// TIA Portal project "Homework-Traffic Light" (V16)

(* hardware
DEVICE "S7-1200 station_1"  S7-1200 Station
   slot 0: "Rack_0"  S7-1200 Rack  Rack  V1.0
   slot 1: "PLC_1"  CPU 1214C DC/DC/DC  6ES7 214-1AG40-0XB0  V4.4
DEVICE "HMI_1"  KTP700 Basic PN
   slot 0: "HMI_1"  KTP700 Basic PN  6AV2 123-2GB03-0AX0  16.0.0.0
   slot 1: "HMI_RT_1"  KTP700 Basic PN  6AV2 123-2GB03-0AX0  16.0.0.0
   slot 5: "HMI_1.IE_CP_1"  PROFINET Interface  16.0.0.0
      slot 1: "PROFINET Interface_1"  PROFINET Interface
         slot 1: "Port_1"  Port
DEVICE "PC-System_1"  SIMATIC PC station
   slot 0: "SIMATIC PC station"  Rail  SIMATIC PC-Station  V1.0
      slot 125: "Stationmanager"  Station_Manager  V6.0.4
   slot 1: "HMI_RT_2"  WinCC RT Advanced  6AV2 104-0xxxx-xxxx  16.0.0.0
      slot 33792: "Computer interface"  Host interface
   slot 2: "IE general_1"  IE General  IE_CP  V8.2.0
*)

// ===== PLC "PLC_1"  CPU 1214C DC/DC/DC =====

VAR_GLOBAL   // PLC tag table "Default tag table"
   "System_Byte" AT %MB8000 : Byte;
   "FirstScan" AT %M8000.0 : Bool;
   "DiagStatusUpdate" AT %M8000.1 : Bool;
   "AlwaysTRUE" AT %M8000.2 : Bool;
   "AlwaysFALSE" AT %M8000.3 : Bool;
   "Clock_Byte" AT %MB8001 : Byte;
   "Clock_10Hz" AT %M8001.0 : Bool;
   "Clock_5Hz" AT %M8001.1 : Bool;
   "Clock_2.5Hz" AT %M8001.2 : Bool;
   "Clock_2Hz" AT %M8001.3 : Bool;
   "Clock_1.25Hz" AT %M8001.4 : Bool;
   "Clock_1Hz" AT %M8001.5 : Bool;
   "Clock_0.625Hz" AT %M8001.6 : Bool;
   "Clock_0.5Hz" AT %M8001.7 : Bool;
   "Pulse1" AT %M0.0 : Bool;
   "Pulse2" AT %M0.1 : Bool;
   "Pulse3" AT %M0.2 : Bool;
   "Pulse4" AT %M0.3 : Bool;
   "Pulse5" AT %M0.4 : Bool;
   "Pulse6" AT %M0.5 : Bool;
   "Pulse_1s" AT %M0.6 : Bool;
   "Pulse7" AT %M0.7 : Bool;
   "Remain3" AT %M1.0 : Bool;
   "Remain1" AT %M1.1 : Bool;
   "Remain2" AT %M1.2 : Bool;
   "Remain4" AT %M1.3 : Bool;
END_VAR

DATA_BLOCK "System Data"   // DB1
{ S7_Optimized_Access := 'TRUE' }
VERSION : 0.1
   VAR
      "Green A" : Bool;
      "Green B" : Bool;
      "Yellow A" : Bool;
      "Yellow B" : Bool;
      "Red A" : Bool;
      "Red B" : Bool;
      HMI_Update : Bool;
      Enable_PP1 : Bool;
      Enalbe_PP2 : Bool;
      Enalbe_PP3 : Bool;
      Start : Bool;
      Stop : Bool;
      RUN_1 : Bool;
      HMI_SET : Bool;
      "Green A _Value" : DInt;
      "Green B_Value" : DInt;
      "Yellow A_value" : DInt;
      "Yellow B_value" : DInt;
      HMI_Green_A : DInt;
      HMI_Green_B : DInt;
      HMI_Yellow_A : DInt;
      HMI_Yellow_B : DInt;
      Cancel : Bool;
      Last_signal : Bool;
      Read_Time : DTL;
      RET_Val : Word;
      Time_day : Bool;
      Time_night : Bool;
   END_VAR
BEGIN
END_DATA_BLOCK

DATA_BLOCK "7SEG_Convert1"   // DB6
{ S7_Optimized_Access := 'TRUE' }
VERSION : 0.1
// stored: InstanceOfName Convert_BCD_7SEG
"Convert_BCD_7SEG"
BEGIN
END_DATA_BLOCK

DATA_BLOCK "Data"   // DB8
{ S7_Optimized_Access := 'TRUE' }
VERSION : 0.1
   VAR
      HMI_Cancel : Bool;
      "Green A _Value" : DInt;
      "Green B_Value" : DInt;
      "1Timer_TImer" : DInt;
      "4Timer_Timer" : DInt;
      Counter_Time : DInt;
      Time_Max_Counter : DInt;
      "Yellow A_Value" : DInt;
      "Yellow B_Value" : DInt;
      "Red A_Value" : DInt;
      "Red B_Value" : DInt;
      "1Timer_Remain_LightB" : DInt;
      "1Timer_Remain_LightA" : DInt;
      TIme_LIGHT_A : DInt;
      Time_LIGHT_B : DInt;
      Timer_Light_YellowB_Remain : DInt;
      Timer_Light_YellowA_Remain : DInt;
      Counter_remain_Light_A : DInt;
      Counter_remain_Light_B : DInt;
      DEC_DIV_A : Int;
      DEC_DIV_B : Int;
      DEC_MOD_A : Int;
      DEC_MOD_B : Int;
      Remain_DEC_A : Int;
      Remain_DEC_B : Int;
      "7SEG_DIV_A" : Byte;
      "7SEG_MOD_A" : Byte;
      "7SEG_DIV_B" : Byte;
      "7SEG_MOD_B" : Byte;
   END_VAR
BEGIN
END_DATA_BLOCK

DATA_BLOCK "7SEG_Convert2"   // DB9
{ S7_Optimized_Access := 'TRUE' }
VERSION : 0.1
// stored: InstanceOfName Convert_BCD_7SEG
"Convert_BCD_7SEG"
BEGIN
END_DATA_BLOCK

DATA_BLOCK "7SEG_Convert3"   // DB10
{ S7_Optimized_Access := 'TRUE' }
VERSION : 0.1
// stored: InstanceOfName Convert_BCD_7SEG
"Convert_BCD_7SEG"
BEGIN
END_DATA_BLOCK

DATA_BLOCK "7SEG_Convert4"   // DB11
{ S7_Optimized_Access := 'TRUE' }
VERSION : 0.1
// stored: InstanceOfName Convert_BCD_7SEG
"Convert_BCD_7SEG"
BEGIN
END_DATA_BLOCK

// folder: System blocks/Program resources

DATA_BLOCK "Timer1"   // DB2
{ S7_Optimized_Access := 'TRUE' }
AUTHOR : Simatic
FAMILY : IEC
NAME : IEC_TMR
VERSION : 1.0
// stored: InstanceOfName IEC_TIMER
"IEC_TIMER"
BEGIN
END_DATA_BLOCK

DATA_BLOCK "Timer2"   // DB3
{ S7_Optimized_Access := 'TRUE' }
AUTHOR : Simatic
FAMILY : IEC
NAME : IEC_TMR
VERSION : 1.0
// stored: InstanceOfName IEC_TIMER
"IEC_TIMER"
BEGIN
END_DATA_BLOCK

DATA_BLOCK "Timer3"   // DB4
{ S7_Optimized_Access := 'TRUE' }
AUTHOR : Simatic
FAMILY : IEC
NAME : IEC_TMR
VERSION : 1.0
// stored: InstanceOfName IEC_TIMER
"IEC_TIMER"
BEGIN
END_DATA_BLOCK

DATA_BLOCK "Timer4"   // DB5
{ S7_Optimized_Access := 'TRUE' }
AUTHOR : Simatic
FAMILY : IEC
NAME : IEC_TMR
VERSION : 1.0
// stored: InstanceOfName IEC_TIMER
"IEC_TIMER"
BEGIN
END_DATA_BLOCK

DATA_BLOCK "T1"   // DB7
{ S7_Optimized_Access := 'TRUE' }
AUTHOR : Simatic
FAMILY : IEC
NAME : IEC_TMR
VERSION : 1.0
// stored: InstanceOfName IEC_TIMER
"IEC_TIMER"
BEGIN
END_DATA_BLOCK

// folder: (top level)

FUNCTION_BLOCK "Convert_BCD_7SEG"   // FB1, SCL
{ S7_Optimized_Access := 'TRUE' }
VERSION : 0.1
   VAR_INPUT
      BCD_Val : Int;
   END_VAR
   VAR_OUTPUT
      "7SEG_Val" : Byte;
   END_VAR
   VAR_TEMP
      tmp : Byte;
   END_VAR
BEGIN
   #tmp := 0;
   IF #BCD_Val =0 THEN
       #tmp := 63;
   END_IF;
   IF #BCD_Val = 1 THEN
       #tmp := 6;
   END_IF;
   IF #BCD_Val = 2 THEN
       #tmp := 91;
   END_IF;
   IF #BCD_Val = 3 THEN
       #tmp := 79;
   END_IF;
   IF #BCD_Val = 4 THEN
       #tmp := 102;
   END_IF;
   IF #BCD_Val = 5 THEN
       #tmp := 109;
   END_IF;
   IF #BCD_Val = 6 THEN
       #tmp := 125;
   END_IF;
   IF #BCD_Val = 7 THEN
       #tmp := 7;
   END_IF;
   IF #BCD_Val = 8 THEN
       #tmp := 127;
   END_IF;
   IF #BCD_Val = 9 THEN
       #tmp := 111;
   END_IF;
   #"7SEG_Val" := #tmp;
END_FUNCTION_BLOCK

FUNCTION "PP2_4Timer" : Void   // FC1, LAD
{ S7_Optimized_Access := 'TRUE' }
VERSION : 0.1
   VAR_TEMP   // added for the SCL form of the ladder/FBD networks
      _w1 : Bool;
   END_VAR
BEGIN

REGION Network 1
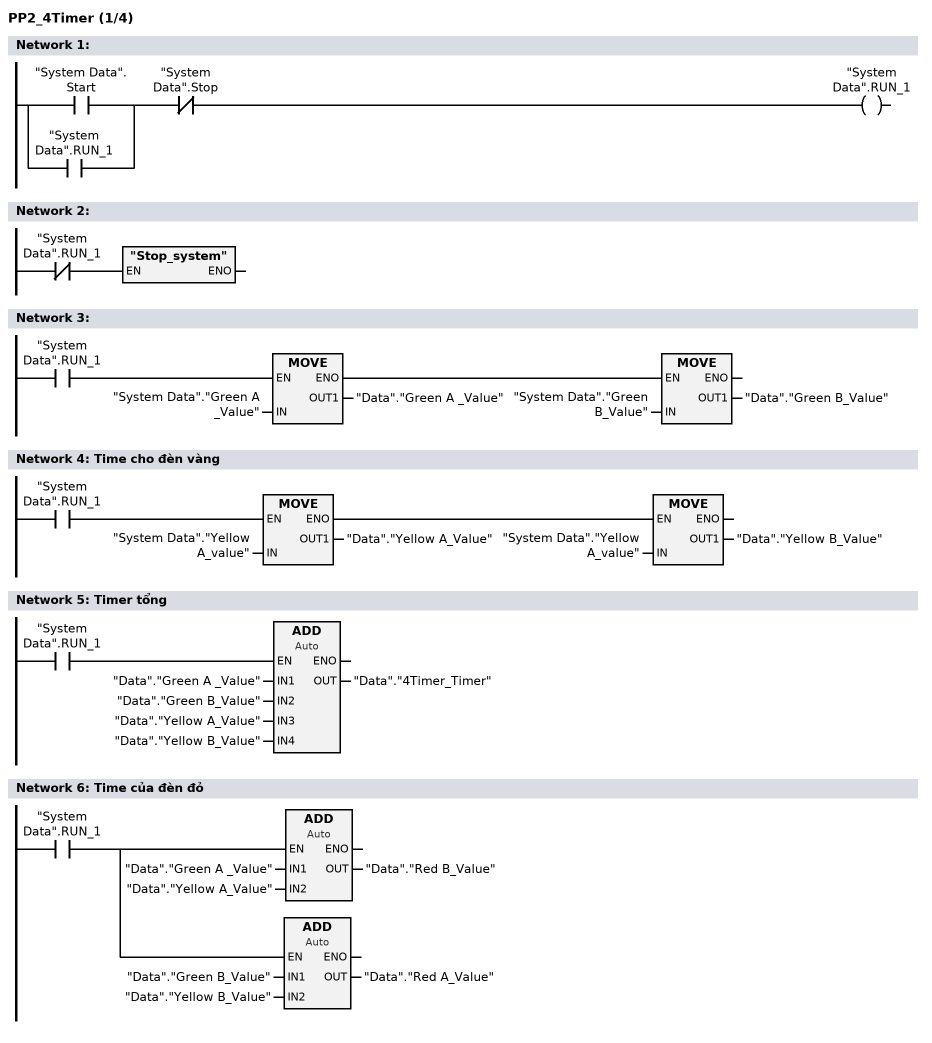
   RUNG wire#powerrail
      Contact( "System Data".Start )
      wire#w1
      I_Contact( "System Data".Stop )
      Coil( "System Data".RUN_1 )
   END_RUNG
   RUNG wire#powerrail
      Contact( "System Data".RUN_1 )
   END_RUNG wire#w1
   // the same network as SCL:
   "System Data".RUN_1 := ("System Data".Start OR "System Data".RUN_1) AND NOT "System Data".Stop;
END_REGION

REGION Network 2
   RUNG wire#powerrail
      I_Contact( "System Data".RUN_1 )
      "Stop_system"()
   END_RUNG
   // the same network as SCL:
   IF NOT "System Data".RUN_1 THEN "Stop_system"(); END_IF;
END_REGION

REGION Network 3
   RUNG wire#powerrail
      Contact( "System Data".RUN_1 )
      Move(in := "System Data"."Green A _Value", out1 => "Data"."Green A _Value")
      Move(in := "System Data"."Green B_Value", out1 => "Data"."Green B_Value")
   END_RUNG
   // the same network as SCL:
   IF "System Data".RUN_1 THEN
       "Data"."Green A _Value" := "System Data"."Green A _Value";
       "Data"."Green B_Value" := "System Data"."Green B_Value";
   END_IF;
END_REGION

REGION Network 4: Time cho đèn vàng
   RUNG wire#powerrail
      Contact( "System Data".RUN_1 )
      Move(in := "System Data"."Yellow A_value", out1 => "Data"."Yellow A_Value")
      Move(in := "System Data"."Yellow A_value", out1 => "Data"."Yellow B_Value")
   END_RUNG
   // the same network as SCL:
   IF "System Data".RUN_1 THEN
       "Data"."Yellow A_Value" := "System Data"."Yellow A_value";
       "Data"."Yellow B_Value" := "System Data"."Yellow A_value";
   END_IF;
END_REGION

REGION Network 5: Timer tổng
   RUNG wire#powerrail
      Contact( "System Data".RUN_1 )
      Add(in1 := "Data"."Green A _Value", in2 := "Data"."Green B_Value", in3 := "Data"."Yellow A_Value", in4 := "Data"."Yellow B_Value", out => "Data"."4Timer_Timer")
   END_RUNG
   // the same network as SCL:
   IF "System Data".RUN_1 THEN
       "Data"."4Timer_Timer" := "Data"."Green A _Value" + "Data"."Green B_Value" + "Data"."Yellow A_Value" + "Data"."Yellow B_Value";
   END_IF;
END_REGION

REGION Network 6: Time của đèn đỏ
   RUNG wire#powerrail
      Contact( "System Data".RUN_1 )
      wire#w1
      Add(in1 := "Data"."Green A _Value", in2 := "Data"."Yellow A_Value", out => "Data"."Red B_Value")
   END_RUNG
   RUNG wire#w1
      Add(in1 := "Data"."Green B_Value", in2 := "Data"."Yellow B_Value", out => "Data"."Red A_Value")
   END_RUNG
   // the same network as SCL:
   IF "System Data".RUN_1 THEN
       "Data"."Red B_Value" := "Data"."Green A _Value" + "Data"."Yellow A_Value";
       "Data"."Red A_Value" := "Data"."Green B_Value" + "Data"."Yellow B_Value";
   END_IF;
END_REGION

REGION Network 7
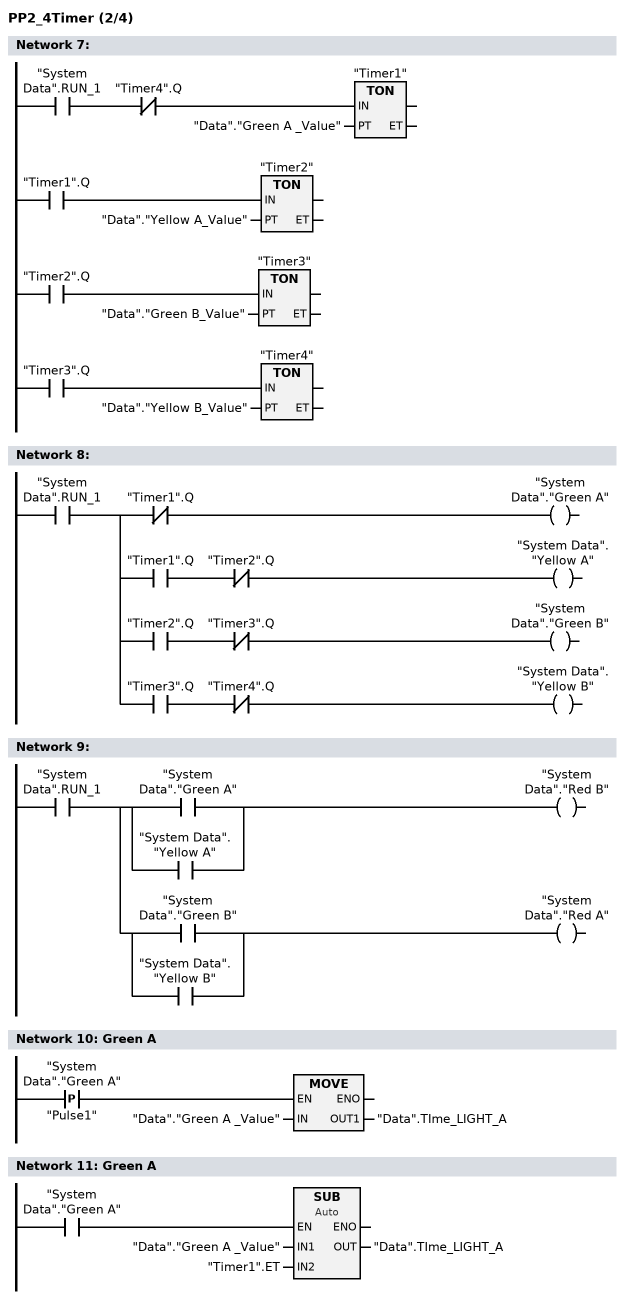
   "Timer1".TON(IN := "System Data".RUN_1 AND NOT "Timer4".Q, PT := "Data"."Green A _Value");
   "Timer2".TON(IN := "Timer1".Q, PT := "Data"."Yellow A_Value");
   "Timer3".TON(IN := "Timer2".Q, PT := "Data"."Green B_Value");
   "Timer4".TON(IN := "Timer3".Q, PT := "Data"."Yellow B_Value");
END_REGION

REGION Network 8
   RUNG wire#powerrail
      Contact( "System Data".RUN_1 )
      wire#w1
      I_Contact( "Timer1".Q )
      Coil( "System Data"."Green A" )
   END_RUNG
   RUNG wire#w1
      Contact( "Timer1".Q )
      I_Contact( "Timer2".Q )
      Coil( "System Data"."Yellow A" )
   END_RUNG
   RUNG wire#w1
      Contact( "Timer2".Q )
      I_Contact( "Timer3".Q )
      Coil( "System Data"."Green B" )
   END_RUNG
   RUNG wire#w1
      Contact( "Timer3".Q )
      I_Contact( "Timer4".Q )
      Coil( "System Data"."Yellow B" )
   END_RUNG
   // the same network as SCL:
   "System Data"."Green A" := "System Data".RUN_1 AND NOT "Timer1".Q;
   "System Data"."Yellow A" := "System Data".RUN_1 AND "Timer1".Q AND NOT "Timer2".Q;
   "System Data"."Green B" := "System Data".RUN_1 AND "Timer2".Q AND NOT "Timer3".Q;
   "System Data"."Yellow B" := "System Data".RUN_1 AND "Timer3".Q AND NOT "Timer4".Q;
END_REGION

REGION Network 9
   RUNG wire#powerrail
      Contact( "System Data".RUN_1 )
      wire#w1
      Contact( "System Data"."Green A" )
      wire#w2
      Coil( "System Data"."Red B" )
   END_RUNG
   RUNG wire#w1
      Contact( "System Data"."Yellow A" )
   END_RUNG wire#w2
   RUNG wire#w1
      Contact( "System Data"."Green B" )
      wire#w3
      Coil( "System Data"."Red A" )
   END_RUNG
   RUNG wire#w1
      Contact( "System Data"."Yellow B" )
   END_RUNG wire#w3
   // the same network as SCL:
   "System Data"."Red B" := "System Data".RUN_1 AND ("System Data"."Green A" OR "System Data"."Yellow A");
   "System Data"."Red A" := "System Data".RUN_1 AND ("System Data"."Green B" OR "System Data"."Yellow B");
END_REGION

REGION Network 10: Green A
   RUNG wire#powerrail
      P_Contact(operand := "System Data"."Green A", bit := "Pulse1")
      Move(in := "Data"."Green A _Value", out1 => "Data".TIme_LIGHT_A)
   END_RUNG
   // the same network as SCL:
   #_w1 := "System Data"."Green A" AND NOT "Pulse1";   // rising edge of "System Data"."Green A"
   "Pulse1" := "System Data"."Green A";
   IF #_w1 THEN "Data".TIme_LIGHT_A := "Data"."Green A _Value"; END_IF;
END_REGION

REGION Network 11: Green A
   RUNG wire#powerrail
      Contact( "System Data"."Green A" )
      Sub(in1 := "Data"."Green A _Value", in2 := "Timer1".ET, out => "Data".TIme_LIGHT_A)
   END_RUNG
   // the same network as SCL:
   IF "System Data"."Green A" THEN "Data".TIme_LIGHT_A := "Data"."Green A _Value" - "Timer1".ET; END_IF;
END_REGION

REGION Network 12: Yellow A
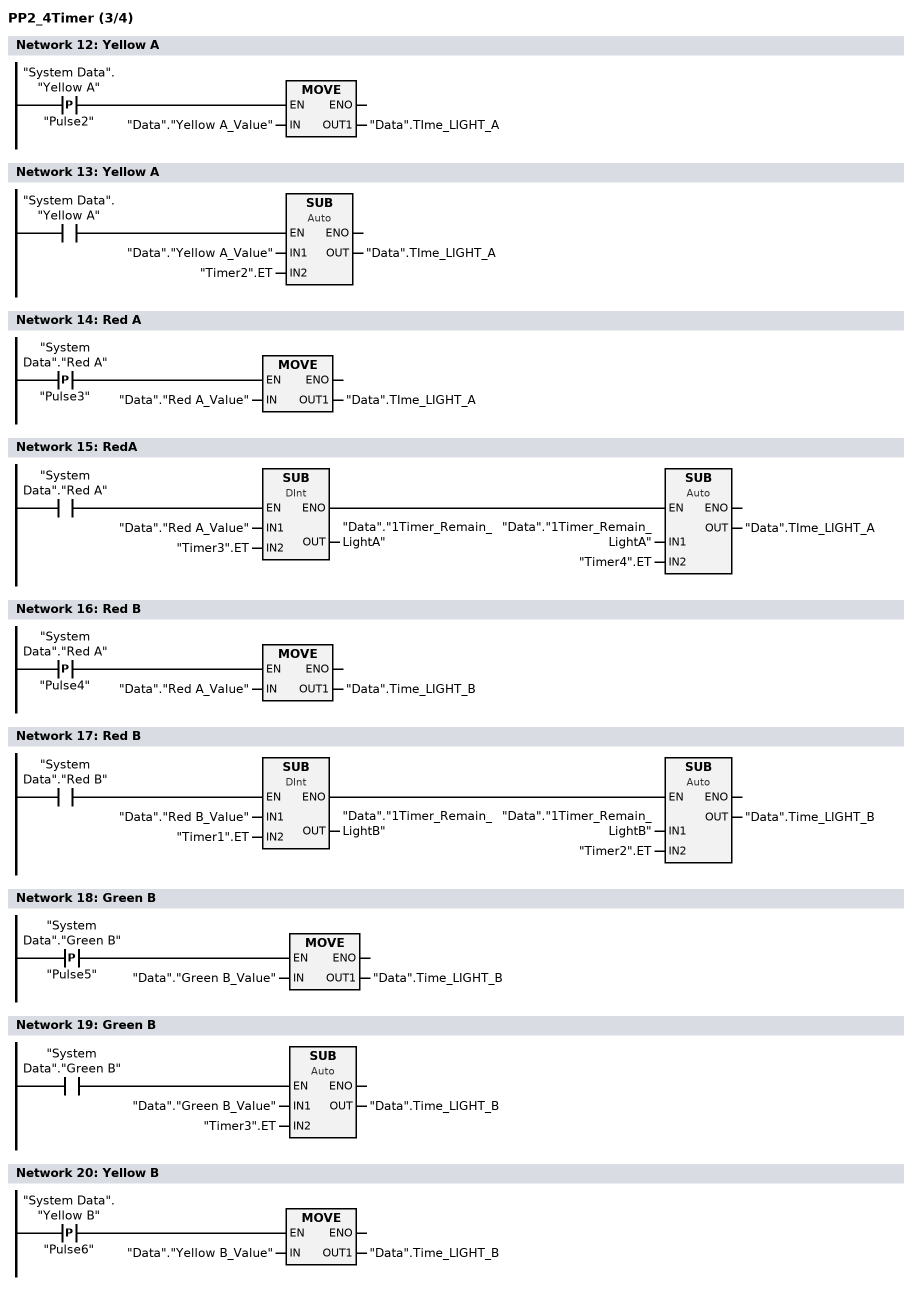
   RUNG wire#powerrail
      P_Contact(operand := "System Data"."Yellow A", bit := "Pulse2")
      Move(in := "Data"."Yellow A_Value", out1 => "Data".TIme_LIGHT_A)
   END_RUNG
   // the same network as SCL:
   #_w1 := "System Data"."Yellow A" AND NOT "Pulse2";   // rising edge of "System Data"."Yellow A"
   "Pulse2" := "System Data"."Yellow A";
   IF #_w1 THEN "Data".TIme_LIGHT_A := "Data"."Yellow A_Value"; END_IF;
END_REGION

REGION Network 13: Yellow A
   RUNG wire#powerrail
      Contact( "System Data"."Yellow A" )
      Sub(in1 := "Data"."Yellow A_Value", in2 := "Timer2".ET, out => "Data".TIme_LIGHT_A)
   END_RUNG
   // the same network as SCL:
   IF "System Data"."Yellow A" THEN "Data".TIme_LIGHT_A := "Data"."Yellow A_Value" - "Timer2".ET; END_IF;
END_REGION

REGION Network 14: Red A
   RUNG wire#powerrail
      P_Contact(operand := "System Data"."Red A", bit := "Pulse3")
      Move(in := "Data"."Red A_Value", out1 => "Data".TIme_LIGHT_A)
   END_RUNG
   // the same network as SCL:
   #_w1 := "System Data"."Red A" AND NOT "Pulse3";   // rising edge of "System Data"."Red A"
   "Pulse3" := "System Data"."Red A";
   IF #_w1 THEN "Data".TIme_LIGHT_A := "Data"."Red A_Value"; END_IF;
END_REGION

REGION Network 15: RedA
   RUNG wire#powerrail
      Contact( "System Data"."Red A" )
      { S7_Templates := "SrcType := DInt" } Sub(in1 := "Data"."Red A_Value", in2 := "Timer3".ET, out => "Data"."1Timer_Remain_LightA")
      Sub(in1 := "Data"."1Timer_Remain_LightA", in2 := "Timer4".ET, out => "Data".TIme_LIGHT_A)
   END_RUNG
   // the same network as SCL:
   IF "System Data"."Red A" THEN
       "Data"."1Timer_Remain_LightA" := "Data"."Red A_Value" - "Timer3".ET;
       "Data".TIme_LIGHT_A := "Data"."1Timer_Remain_LightA" - "Timer4".ET;
   END_IF;
END_REGION

REGION Network 16: Red B
   RUNG wire#powerrail
      P_Contact(operand := "System Data"."Red A", bit := "Pulse4")
      Move(in := "Data"."Red A_Value", out1 => "Data".Time_LIGHT_B)
   END_RUNG
   // the same network as SCL:
   #_w1 := "System Data"."Red A" AND NOT "Pulse4";   // rising edge of "System Data"."Red A"
   "Pulse4" := "System Data"."Red A";
   IF #_w1 THEN "Data".Time_LIGHT_B := "Data"."Red A_Value"; END_IF;
END_REGION

REGION Network 17: Red B
   RUNG wire#powerrail
      Contact( "System Data"."Red B" )
      { S7_Templates := "SrcType := DInt" } Sub(in1 := "Data"."Red B_Value", in2 := "Timer1".ET, out => "Data"."1Timer_Remain_LightB")
      Sub(in1 := "Data"."1Timer_Remain_LightB", in2 := "Timer2".ET, out => "Data".Time_LIGHT_B)
   END_RUNG
   // the same network as SCL:
   IF "System Data"."Red B" THEN
       "Data"."1Timer_Remain_LightB" := "Data"."Red B_Value" - "Timer1".ET;
       "Data".Time_LIGHT_B := "Data"."1Timer_Remain_LightB" - "Timer2".ET;
   END_IF;
END_REGION

REGION Network 18: Green B
   RUNG wire#powerrail
      P_Contact(operand := "System Data"."Green B", bit := "Pulse5")
      Move(in := "Data"."Green B_Value", out1 => "Data".Time_LIGHT_B)
   END_RUNG
   // the same network as SCL:
   #_w1 := "System Data"."Green B" AND NOT "Pulse5";   // rising edge of "System Data"."Green B"
   "Pulse5" := "System Data"."Green B";
   IF #_w1 THEN "Data".Time_LIGHT_B := "Data"."Green B_Value"; END_IF;
END_REGION

REGION Network 19: Green B
   RUNG wire#powerrail
      Contact( "System Data"."Green B" )
      Sub(in1 := "Data"."Green B_Value", in2 := "Timer3".ET, out => "Data".Time_LIGHT_B)
   END_RUNG
   // the same network as SCL:
   IF "System Data"."Green B" THEN "Data".Time_LIGHT_B := "Data"."Green B_Value" - "Timer3".ET; END_IF;
END_REGION

REGION Network 20: Yellow B
   RUNG wire#powerrail
      P_Contact(operand := "System Data"."Yellow B", bit := "Pulse6")
      Move(in := "Data"."Yellow B_Value", out1 => "Data".Time_LIGHT_B)
   END_RUNG
   // the same network as SCL:
   #_w1 := "System Data"."Yellow B" AND NOT "Pulse6";   // rising edge of "System Data"."Yellow B"
   "Pulse6" := "System Data"."Yellow B";
   IF #_w1 THEN "Data".Time_LIGHT_B := "Data"."Yellow B_Value"; END_IF;
END_REGION

REGION Network 21: Yellow B
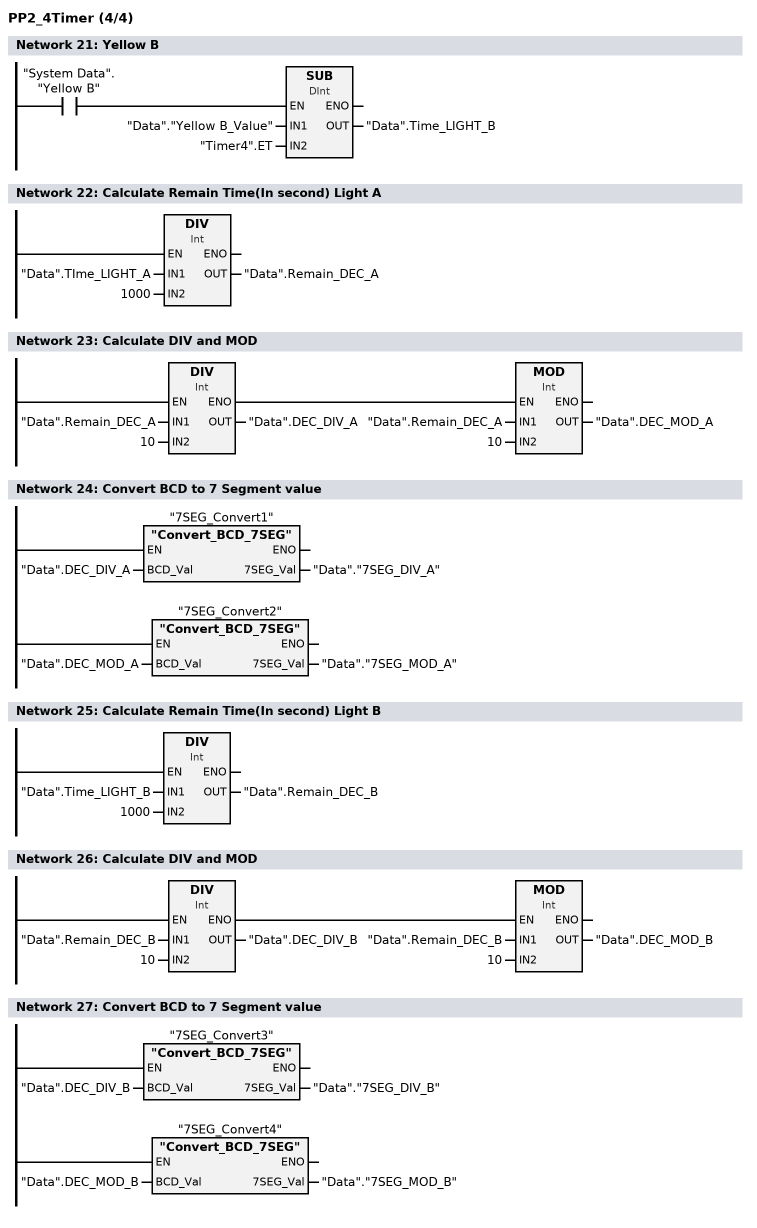
   RUNG wire#powerrail
      Contact( "System Data"."Yellow B" )
      { S7_Templates := "SrcType := DInt" } Sub(in1 := "Data"."Yellow B_Value", in2 := "Timer4".ET, out => "Data".Time_LIGHT_B)
   END_RUNG
   // the same network as SCL:
   IF "System Data"."Yellow B" THEN "Data".Time_LIGHT_B := "Data"."Yellow B_Value" - "Timer4".ET; END_IF;
END_REGION

REGION Network 22: Calculate Remain Time(In second) Light A
   RUNG wire#powerrail
      { S7_Templates := "SrcType := Int" } Div(in1 := "Data".TIme_LIGHT_A, in2 := 1000, out => "Data".Remain_DEC_A)
   END_RUNG
   // the same network as SCL:
   "Data".Remain_DEC_A := "Data".TIme_LIGHT_A / 1000;
END_REGION

REGION Network 23: Calculate DIV and MOD
   RUNG wire#powerrail
      { S7_Templates := "SrcType := Int" } Div(in1 := "Data".Remain_DEC_A, in2 := 10, out => "Data".DEC_DIV_A)
      { S7_Templates := "SrcType := Int" } Mod(in1 := "Data".Remain_DEC_A, in2 := 10, out => "Data".DEC_MOD_A)
   END_RUNG
   // the same network as SCL:
   "Data".DEC_DIV_A := "Data".Remain_DEC_A / 10;
   "Data".DEC_MOD_A := "Data".Remain_DEC_A MOD 10;
END_REGION

REGION Network 24: Convert BCD to 7 Segment value
   RUNG wire#powerrail
      "7SEG_Convert1"(BCD_Val := "Data".DEC_DIV_A, "7SEG_Val" => "Data"."7SEG_DIV_A")
   END_RUNG
   RUNG wire#powerrail
      "7SEG_Convert2"(BCD_Val := "Data".DEC_MOD_A, "7SEG_Val" => "Data"."7SEG_MOD_A")
   END_RUNG
   // the same network as SCL:
   "7SEG_Convert1"(BCD_Val := "Data".DEC_DIV_A, "7SEG_Val" => "Data"."7SEG_DIV_A");   // "Convert_BCD_7SEG"
   "7SEG_Convert2"(BCD_Val := "Data".DEC_MOD_A, "7SEG_Val" => "Data"."7SEG_MOD_A");   // "Convert_BCD_7SEG"
END_REGION

REGION Network 25: Calculate Remain Time(In second) Light B
   RUNG wire#powerrail
      { S7_Templates := "SrcType := Int" } Div(in1 := "Data".Time_LIGHT_B, in2 := 1000, out => "Data".Remain_DEC_B)
   END_RUNG
   // the same network as SCL:
   "Data".Remain_DEC_B := "Data".Time_LIGHT_B / 1000;
END_REGION

REGION Network 26: Calculate DIV and MOD
   RUNG wire#powerrail
      { S7_Templates := "SrcType := Int" } Div(in1 := "Data".Remain_DEC_B, in2 := 10, out => "Data".DEC_DIV_B)
      { S7_Templates := "SrcType := Int" } Mod(in1 := "Data".Remain_DEC_B, in2 := 10, out => "Data".DEC_MOD_B)
   END_RUNG
   // the same network as SCL:
   "Data".DEC_DIV_B := "Data".Remain_DEC_B / 10;
   "Data".DEC_MOD_B := "Data".Remain_DEC_B MOD 10;
END_REGION

REGION Network 27: Convert BCD to 7 Segment value
   RUNG wire#powerrail
      "7SEG_Convert3"(BCD_Val := "Data".DEC_DIV_B, "7SEG_Val" => "Data"."7SEG_DIV_B")
   END_RUNG
   RUNG wire#powerrail
      "7SEG_Convert4"(BCD_Val := "Data".DEC_MOD_B, "7SEG_Val" => "Data"."7SEG_MOD_B")
   END_RUNG
   // the same network as SCL:
   "7SEG_Convert3"(BCD_Val := "Data".DEC_DIV_B, "7SEG_Val" => "Data"."7SEG_DIV_B");   // "Convert_BCD_7SEG"
   "7SEG_Convert4"(BCD_Val := "Data".DEC_MOD_B, "7SEG_Val" => "Data"."7SEG_MOD_B");   // "Convert_BCD_7SEG"
END_REGION
END_FUNCTION

FUNCTION "PP1_1Timer" : Void   // FC2, LAD
{ S7_Optimized_Access := 'TRUE' }
VERSION : 0.1
   VAR_TEMP   // added for the SCL form of the ladder/FBD networks
      _w1 : Bool;
   END_VAR
BEGIN

REGION Network 1
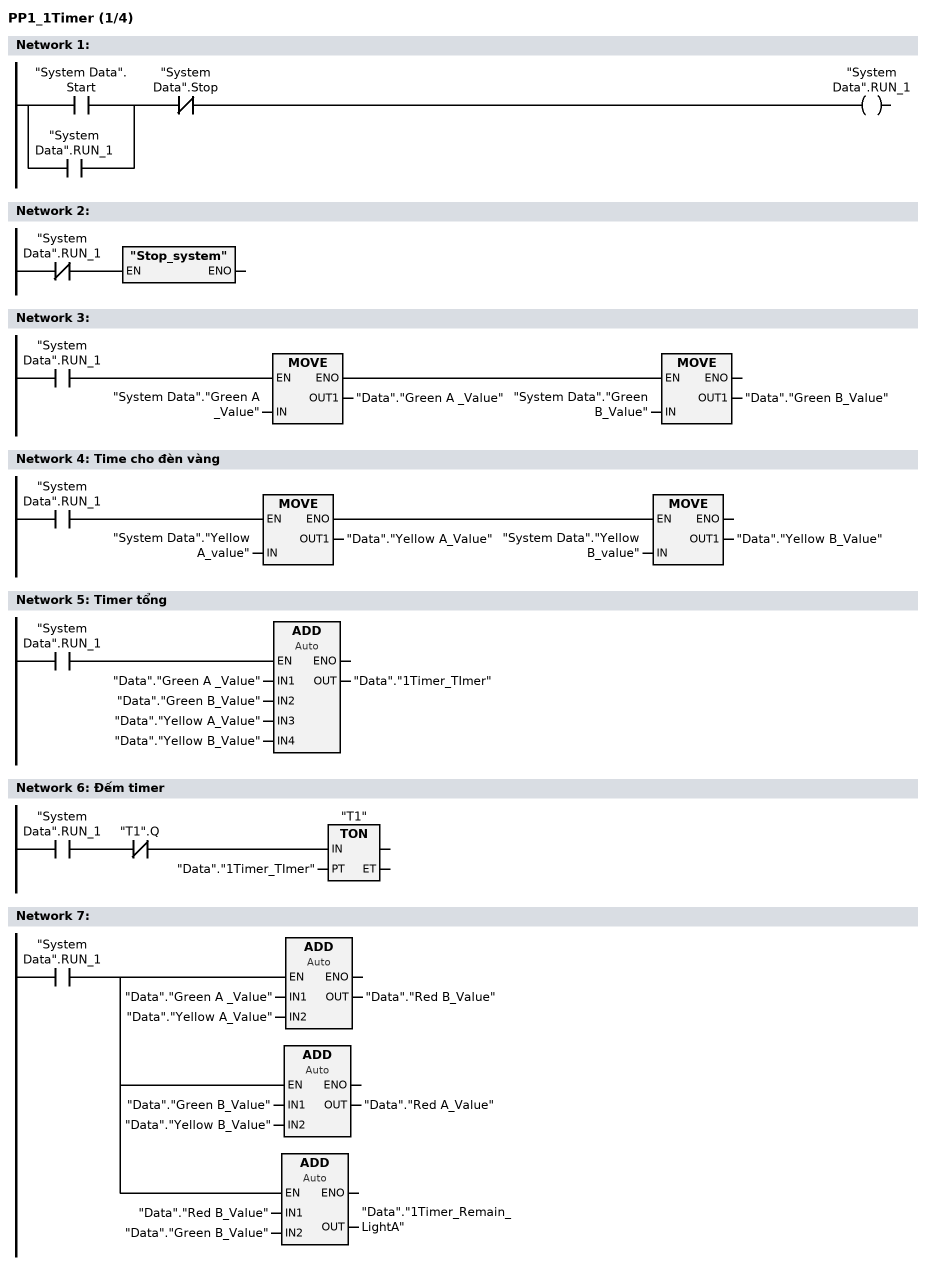
   RUNG wire#powerrail
      Contact( "System Data".Start )
      wire#w1
      I_Contact( "System Data".Stop )
      Coil( "System Data".RUN_1 )
   END_RUNG
   RUNG wire#powerrail
      Contact( "System Data".RUN_1 )
   END_RUNG wire#w1
   // the same network as SCL:
   "System Data".RUN_1 := ("System Data".Start OR "System Data".RUN_1) AND NOT "System Data".Stop;
END_REGION

REGION Network 2
   RUNG wire#powerrail
      I_Contact( "System Data".RUN_1 )
      "Stop_system"()
   END_RUNG
   // the same network as SCL:
   IF NOT "System Data".RUN_1 THEN "Stop_system"(); END_IF;
END_REGION

REGION Network 3
   RUNG wire#powerrail
      Contact( "System Data".RUN_1 )
      Move(in := "System Data"."Green A _Value", out1 => "Data"."Green A _Value")
      Move(in := "System Data"."Green B_Value", out1 => "Data"."Green B_Value")
   END_RUNG
   // the same network as SCL:
   IF "System Data".RUN_1 THEN
       "Data"."Green A _Value" := "System Data"."Green A _Value";
       "Data"."Green B_Value" := "System Data"."Green B_Value";
   END_IF;
END_REGION

REGION Network 4: Time cho đèn vàng
   RUNG wire#powerrail
      Contact( "System Data".RUN_1 )
      Move(in := "System Data"."Yellow A_value", out1 => "Data"."Yellow A_Value")
      Move(in := "System Data"."Yellow B_value", out1 => "Data"."Yellow B_Value")
   END_RUNG
   // the same network as SCL:
   IF "System Data".RUN_1 THEN
       "Data"."Yellow A_Value" := "System Data"."Yellow A_value";
       "Data"."Yellow B_Value" := "System Data"."Yellow B_value";
   END_IF;
END_REGION

REGION Network 5: Timer tổng
   RUNG wire#powerrail
      Contact( "System Data".RUN_1 )
      Add(in1 := "Data"."Green A _Value", in2 := "Data"."Green B_Value", in3 := "Data"."Yellow A_Value", in4 := "Data"."Yellow B_Value", out => "Data"."1Timer_TImer")
   END_RUNG
   // the same network as SCL:
   IF "System Data".RUN_1 THEN
       "Data"."1Timer_TImer" := "Data"."Green A _Value" + "Data"."Green B_Value" + "Data"."Yellow A_Value" + "Data"."Yellow B_Value";
   END_IF;
END_REGION

REGION Network 6: Đếm timer
   "T1".TON(IN := "System Data".RUN_1 AND NOT "T1".Q, PT := "Data"."1Timer_TImer");
END_REGION

REGION Network 7
   RUNG wire#powerrail
      Contact( "System Data".RUN_1 )
      wire#w1
      Add(in1 := "Data"."Green A _Value", in2 := "Data"."Yellow A_Value", out => "Data"."Red B_Value")
   END_RUNG
   RUNG wire#w1
      Add(in1 := "Data"."Green B_Value", in2 := "Data"."Yellow B_Value", out => "Data"."Red A_Value")
   END_RUNG
   RUNG wire#w1
      Add(in1 := "Data"."Red B_Value", in2 := "Data"."Green B_Value", out => "Data"."1Timer_Remain_LightA")
   END_RUNG
   // the same network as SCL:
   IF "System Data".RUN_1 THEN
       "Data"."Red B_Value" := "Data"."Green A _Value" + "Data"."Yellow A_Value";
       "Data"."Red A_Value" := "Data"."Green B_Value" + "Data"."Yellow B_Value";
       "Data"."1Timer_Remain_LightA" := "Data"."Red B_Value" + "Data"."Green B_Value";
   END_IF;
END_REGION

REGION Network 8
   // 5s đèn xanh
   // 5
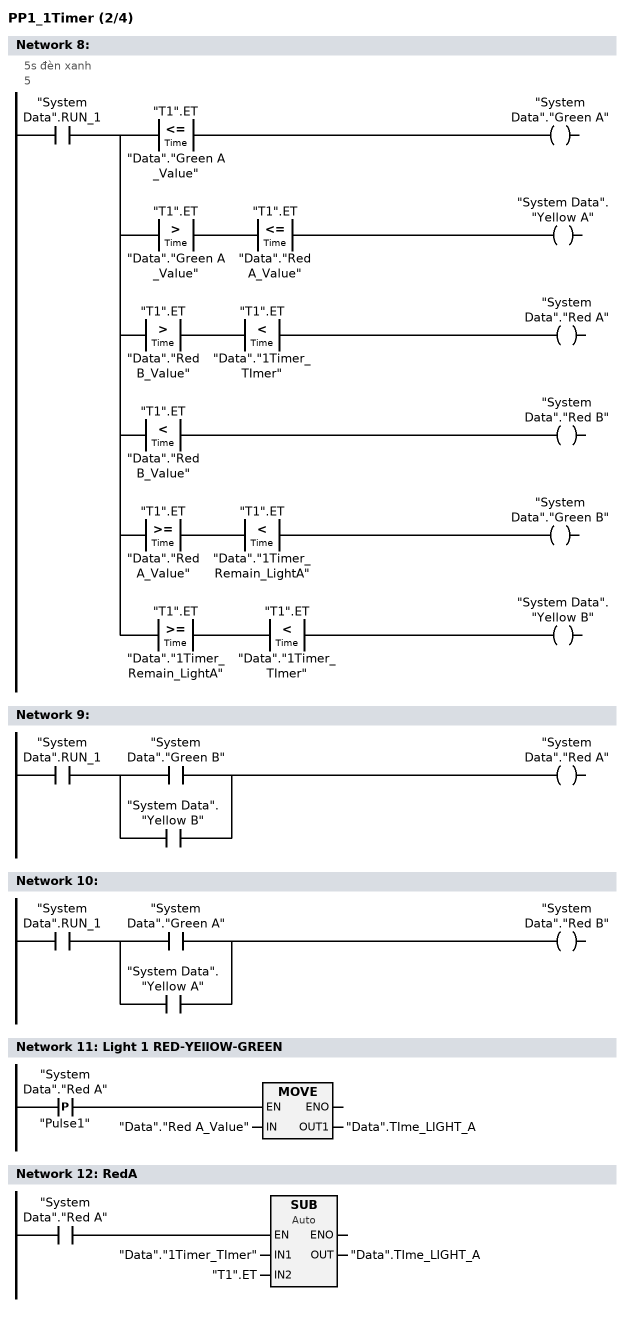
   RUNG wire#powerrail
      Contact( "System Data".RUN_1 )
      wire#w1
      { S7_Templates := "SrcType := Time" } LE_Contact(in1 := "T1".ET, in2 := "Data"."Green A _Value")
      Coil( "System Data"."Green A" )
   END_RUNG
   RUNG wire#w1
      { S7_Templates := "SrcType := Time" } GT_Contact(in1 := "T1".ET, in2 := "Data"."Green A _Value")
      { S7_Templates := "SrcType := Time" } LE_Contact(in1 := "T1".ET, in2 := "Data"."Red A_Value")
      Coil( "System Data"."Yellow A" )
   END_RUNG
   RUNG wire#w1
      { S7_Templates := "SrcType := Time" } GT_Contact(in1 := "T1".ET, in2 := "Data"."Red B_Value")
      { S7_Templates := "SrcType := Time" } LT_Contact(in1 := "T1".ET, in2 := "Data"."1Timer_TImer")
      Coil( "System Data"."Red A" )
   END_RUNG
   RUNG wire#w1
      { S7_Templates := "SrcType := Time" } LT_Contact(in1 := "T1".ET, in2 := "Data"."Red B_Value")
      Coil( "System Data"."Red B" )
   END_RUNG
   RUNG wire#w1
      { S7_Templates := "SrcType := Time" } GE_Contact(in1 := "T1".ET, in2 := "Data"."Red A_Value")
      { S7_Templates := "SrcType := Time" } LT_Contact(in1 := "T1".ET, in2 := "Data"."1Timer_Remain_LightA")
      Coil( "System Data"."Green B" )
   END_RUNG
   RUNG wire#w1
      { S7_Templates := "SrcType := Time" } GE_Contact(in1 := "T1".ET, in2 := "Data"."1Timer_Remain_LightA")
      { S7_Templates := "SrcType := Time" } LT_Contact(in1 := "T1".ET, in2 := "Data"."1Timer_TImer")
      Coil( "System Data"."Yellow B" )
   END_RUNG
   // the same network as SCL:
   "System Data"."Green A" := "System Data".RUN_1 AND ("T1".ET <= "Data"."Green A _Value");
   "System Data"."Yellow A" := "System Data".RUN_1 AND ("T1".ET > "Data"."Green A _Value") AND ("T1".ET <= "Data"."Red A_Value");
   "System Data"."Red A" := "System Data".RUN_1 AND ("T1".ET > "Data"."Red B_Value") AND ("T1".ET < "Data"."1Timer_TImer");
   "System Data"."Red B" := "System Data".RUN_1 AND ("T1".ET < "Data"."Red B_Value");
   "System Data"."Green B" := "System Data".RUN_1 AND ("T1".ET >= "Data"."Red A_Value") AND ("T1".ET < "Data"."1Timer_Remain_LightA");
   "System Data"."Yellow B" := "System Data".RUN_1 AND ("T1".ET >= "Data"."1Timer_Remain_LightA") AND ("T1".ET < "Data"."1Timer_TImer");
END_REGION

REGION Network 9
   RUNG wire#powerrail
      Contact( "System Data".RUN_1 )
      wire#w1
      Contact( "System Data"."Green B" )
      wire#w2
      Coil( "System Data"."Red A" )
   END_RUNG
   RUNG wire#w1
      Contact( "System Data"."Yellow B" )
   END_RUNG wire#w2
   // the same network as SCL:
   "System Data"."Red A" := "System Data".RUN_1 AND ("System Data"."Green B" OR "System Data"."Yellow B");
END_REGION

REGION Network 10
   RUNG wire#powerrail
      Contact( "System Data".RUN_1 )
      wire#w1
      Contact( "System Data"."Green A" )
      wire#w2
      Coil( "System Data"."Red B" )
   END_RUNG
   RUNG wire#w1
      Contact( "System Data"."Yellow A" )
   END_RUNG wire#w2
   // the same network as SCL:
   "System Data"."Red B" := "System Data".RUN_1 AND ("System Data"."Green A" OR "System Data"."Yellow A");
END_REGION

REGION Network 11: Light 1 RED-YEllOW-GREEN
   RUNG wire#powerrail
      P_Contact(operand := "System Data"."Red A", bit := "Pulse1")
      Move(in := "Data"."Red A_Value", out1 => "Data".TIme_LIGHT_A)
   END_RUNG
   // the same network as SCL:
   #_w1 := "System Data"."Red A" AND NOT "Pulse1";   // rising edge of "System Data"."Red A"
   "Pulse1" := "System Data"."Red A";
   IF #_w1 THEN "Data".TIme_LIGHT_A := "Data"."Red A_Value"; END_IF;
END_REGION

REGION Network 12: RedA
   RUNG wire#powerrail
      Contact( "System Data"."Red A" )
      Sub(in1 := "Data"."1Timer_TImer", in2 := "T1".ET, out => "Data".TIme_LIGHT_A)
   END_RUNG
   // the same network as SCL:
   IF "System Data"."Red A" THEN "Data".TIme_LIGHT_A := "Data"."1Timer_TImer" - "T1".ET; END_IF;
END_REGION

REGION Network 13
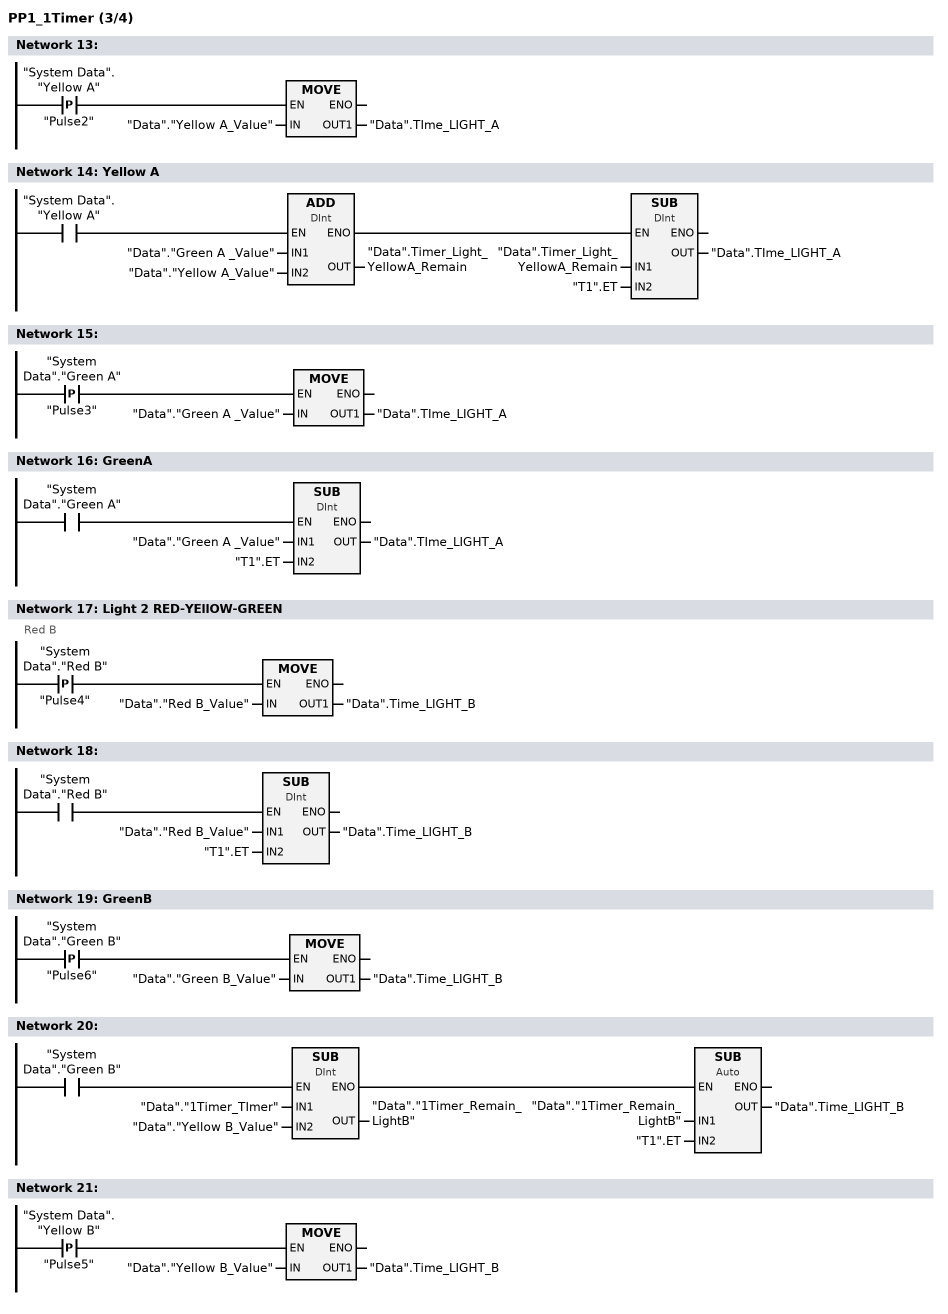
   RUNG wire#powerrail
      P_Contact(operand := "System Data"."Yellow A", bit := "Pulse2")
      Move(in := "Data"."Yellow A_Value", out1 => "Data".TIme_LIGHT_A)
   END_RUNG
   // the same network as SCL:
   #_w1 := "System Data"."Yellow A" AND NOT "Pulse2";   // rising edge of "System Data"."Yellow A"
   "Pulse2" := "System Data"."Yellow A";
   IF #_w1 THEN "Data".TIme_LIGHT_A := "Data"."Yellow A_Value"; END_IF;
END_REGION

REGION Network 14: Yellow A
   RUNG wire#powerrail
      Contact( "System Data"."Yellow A" )
      { S7_Templates := "SrcType := DInt" } Add(in1 := "Data"."Green A _Value", in2 := "Data"."Yellow A_Value", out => "Data".Timer_Light_YellowA_Remain)
      { S7_Templates := "SrcType := DInt" } Sub(in1 := "Data".Timer_Light_YellowA_Remain, in2 := "T1".ET, out => "Data".TIme_LIGHT_A)
   END_RUNG
   // the same network as SCL:
   IF "System Data"."Yellow A" THEN
       "Data".Timer_Light_YellowA_Remain := "Data"."Green A _Value" + "Data"."Yellow A_Value";
       "Data".TIme_LIGHT_A := "Data".Timer_Light_YellowA_Remain - "T1".ET;
   END_IF;
END_REGION

REGION Network 15
   RUNG wire#powerrail
      P_Contact(operand := "System Data"."Green A", bit := "Pulse3")
      Move(in := "Data"."Green A _Value", out1 => "Data".TIme_LIGHT_A)
   END_RUNG
   // the same network as SCL:
   #_w1 := "System Data"."Green A" AND NOT "Pulse3";   // rising edge of "System Data"."Green A"
   "Pulse3" := "System Data"."Green A";
   IF #_w1 THEN "Data".TIme_LIGHT_A := "Data"."Green A _Value"; END_IF;
END_REGION

REGION Network 16: GreenA
   RUNG wire#powerrail
      Contact( "System Data"."Green A" )
      { S7_Templates := "SrcType := DInt" } Sub(in1 := "Data"."Green A _Value", in2 := "T1".ET, out => "Data".TIme_LIGHT_A)
   END_RUNG
   // the same network as SCL:
   IF "System Data"."Green A" THEN "Data".TIme_LIGHT_A := "Data"."Green A _Value" - "T1".ET; END_IF;
END_REGION

REGION Network 17: Light 2 RED-YEllOW-GREEN
   // Red B
   RUNG wire#powerrail
      P_Contact(operand := "System Data"."Red B", bit := "Pulse4")
      Move(in := "Data"."Red B_Value", out1 => "Data".Time_LIGHT_B)
   END_RUNG
   // the same network as SCL:
   #_w1 := "System Data"."Red B" AND NOT "Pulse4";   // rising edge of "System Data"."Red B"
   "Pulse4" := "System Data"."Red B";
   IF #_w1 THEN "Data".Time_LIGHT_B := "Data"."Red B_Value"; END_IF;
END_REGION

REGION Network 18
   RUNG wire#powerrail
      Contact( "System Data"."Red B" )
      { S7_Templates := "SrcType := DInt" } Sub(in1 := "Data"."Red B_Value", in2 := "T1".ET, out => "Data".Time_LIGHT_B)
   END_RUNG
   // the same network as SCL:
   IF "System Data"."Red B" THEN "Data".Time_LIGHT_B := "Data"."Red B_Value" - "T1".ET; END_IF;
END_REGION

REGION Network 19: GreenB
   RUNG wire#powerrail
      P_Contact(operand := "System Data"."Green B", bit := "Pulse6")
      Move(in := "Data"."Green B_Value", out1 => "Data".Time_LIGHT_B)
   END_RUNG
   // the same network as SCL:
   #_w1 := "System Data"."Green B" AND NOT "Pulse6";   // rising edge of "System Data"."Green B"
   "Pulse6" := "System Data"."Green B";
   IF #_w1 THEN "Data".Time_LIGHT_B := "Data"."Green B_Value"; END_IF;
END_REGION

REGION Network 20
   RUNG wire#powerrail
      Contact( "System Data"."Green B" )
      { S7_Templates := "SrcType := DInt" } Sub(in1 := "Data"."1Timer_TImer", in2 := "Data"."Yellow B_Value", out => "Data"."1Timer_Remain_LightB")
      Sub(in1 := "Data"."1Timer_Remain_LightB", in2 := "T1".ET, out => "Data".Time_LIGHT_B)
   END_RUNG
   // the same network as SCL:
   IF "System Data"."Green B" THEN
       "Data"."1Timer_Remain_LightB" := "Data"."1Timer_TImer" - "Data"."Yellow B_Value";
       "Data".Time_LIGHT_B := "Data"."1Timer_Remain_LightB" - "T1".ET;
   END_IF;
END_REGION

REGION Network 21
   RUNG wire#powerrail
      P_Contact(operand := "System Data"."Yellow B", bit := "Pulse5")
      Move(in := "Data"."Yellow B_Value", out1 => "Data".Time_LIGHT_B)
   END_RUNG
   // the same network as SCL:
   #_w1 := "System Data"."Yellow B" AND NOT "Pulse5";   // rising edge of "System Data"."Yellow B"
   "Pulse5" := "System Data"."Yellow B";
   IF #_w1 THEN "Data".Time_LIGHT_B := "Data"."Yellow B_Value"; END_IF;
END_REGION

REGION Network 22: Yellow B
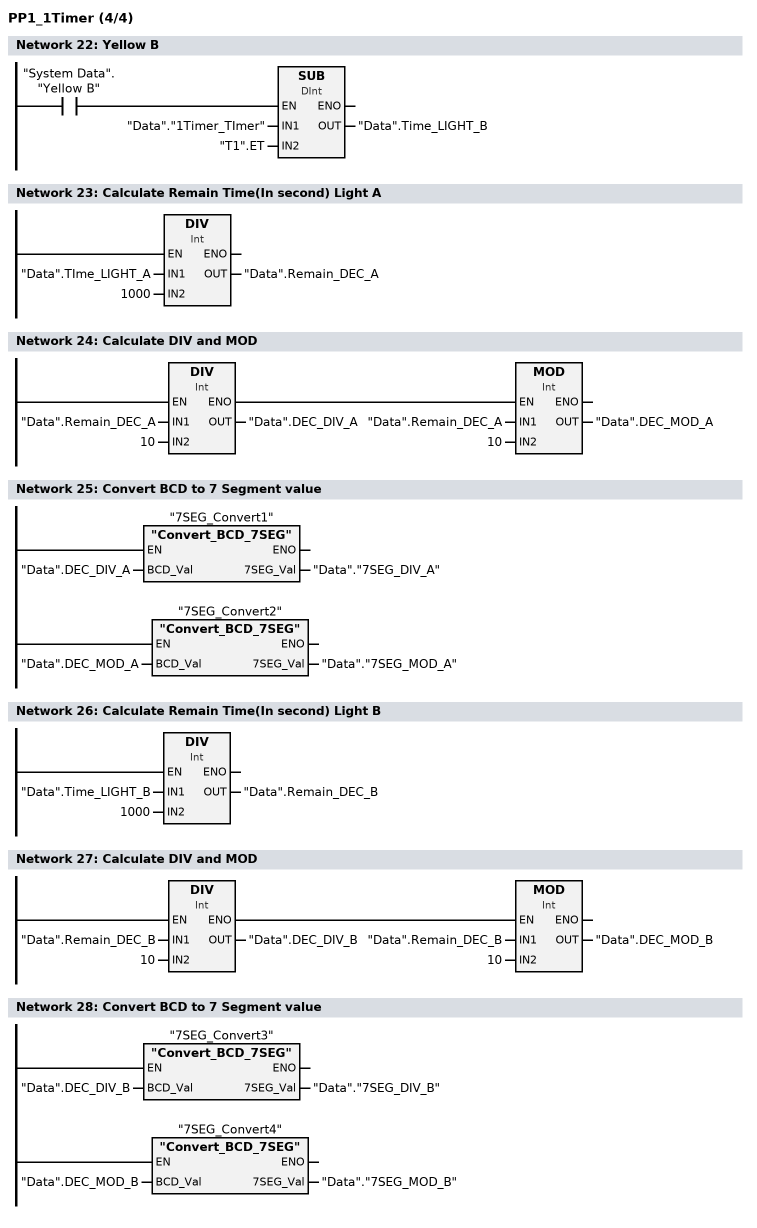
   RUNG wire#powerrail
      Contact( "System Data"."Yellow B" )
      { S7_Templates := "SrcType := DInt" } Sub(in1 := "Data"."1Timer_TImer", in2 := "T1".ET, out => "Data".Time_LIGHT_B)
   END_RUNG
   // the same network as SCL:
   IF "System Data"."Yellow B" THEN "Data".Time_LIGHT_B := "Data"."1Timer_TImer" - "T1".ET; END_IF;
END_REGION

REGION Network 23: Calculate Remain Time(In second) Light A
   RUNG wire#powerrail
      { S7_Templates := "SrcType := Int" } Div(in1 := "Data".TIme_LIGHT_A, in2 := 1000, out => "Data".Remain_DEC_A)
   END_RUNG
   // the same network as SCL:
   "Data".Remain_DEC_A := "Data".TIme_LIGHT_A / 1000;
END_REGION

REGION Network 24: Calculate DIV and MOD
   RUNG wire#powerrail
      { S7_Templates := "SrcType := Int" } Div(in1 := "Data".Remain_DEC_A, in2 := 10, out => "Data".DEC_DIV_A)
      { S7_Templates := "SrcType := Int" } Mod(in1 := "Data".Remain_DEC_A, in2 := 10, out => "Data".DEC_MOD_A)
   END_RUNG
   // the same network as SCL:
   "Data".DEC_DIV_A := "Data".Remain_DEC_A / 10;
   "Data".DEC_MOD_A := "Data".Remain_DEC_A MOD 10;
END_REGION

REGION Network 25: Convert BCD to 7 Segment value
   RUNG wire#powerrail
      "7SEG_Convert1"(BCD_Val := "Data".DEC_DIV_A, "7SEG_Val" => "Data"."7SEG_DIV_A")
   END_RUNG
   RUNG wire#powerrail
      "7SEG_Convert2"(BCD_Val := "Data".DEC_MOD_A, "7SEG_Val" => "Data"."7SEG_MOD_A")
   END_RUNG
   // the same network as SCL:
   "7SEG_Convert1"(BCD_Val := "Data".DEC_DIV_A, "7SEG_Val" => "Data"."7SEG_DIV_A");   // "Convert_BCD_7SEG"
   "7SEG_Convert2"(BCD_Val := "Data".DEC_MOD_A, "7SEG_Val" => "Data"."7SEG_MOD_A");   // "Convert_BCD_7SEG"
END_REGION

REGION Network 26: Calculate Remain Time(In second) Light B
   RUNG wire#powerrail
      { S7_Templates := "SrcType := Int" } Div(in1 := "Data".Time_LIGHT_B, in2 := 1000, out => "Data".Remain_DEC_B)
   END_RUNG
   // the same network as SCL:
   "Data".Remain_DEC_B := "Data".Time_LIGHT_B / 1000;
END_REGION

REGION Network 27: Calculate DIV and MOD
   RUNG wire#powerrail
      { S7_Templates := "SrcType := Int" } Div(in1 := "Data".Remain_DEC_B, in2 := 10, out => "Data".DEC_DIV_B)
      { S7_Templates := "SrcType := Int" } Mod(in1 := "Data".Remain_DEC_B, in2 := 10, out => "Data".DEC_MOD_B)
   END_RUNG
   // the same network as SCL:
   "Data".DEC_DIV_B := "Data".Remain_DEC_B / 10;
   "Data".DEC_MOD_B := "Data".Remain_DEC_B MOD 10;
END_REGION

REGION Network 28: Convert BCD to 7 Segment value
   RUNG wire#powerrail
      "7SEG_Convert3"(BCD_Val := "Data".DEC_DIV_B, "7SEG_Val" => "Data"."7SEG_DIV_B")
   END_RUNG
   RUNG wire#powerrail
      "7SEG_Convert4"(BCD_Val := "Data".DEC_MOD_B, "7SEG_Val" => "Data"."7SEG_MOD_B")
   END_RUNG
   // the same network as SCL:
   "7SEG_Convert3"(BCD_Val := "Data".DEC_DIV_B, "7SEG_Val" => "Data"."7SEG_DIV_B");   // "Convert_BCD_7SEG"
   "7SEG_Convert4"(BCD_Val := "Data".DEC_MOD_B, "7SEG_Val" => "Data"."7SEG_MOD_B");   // "Convert_BCD_7SEG"
END_REGION
END_FUNCTION

FUNCTION "PP3_Counter" : Void   // FC3, LAD
{ S7_Optimized_Access := 'TRUE' }
VERSION : 0.1
   VAR_TEMP   // added for the SCL form of the ladder/FBD networks
      _w1 : Bool;
   END_VAR
BEGIN

REGION Network 1: System
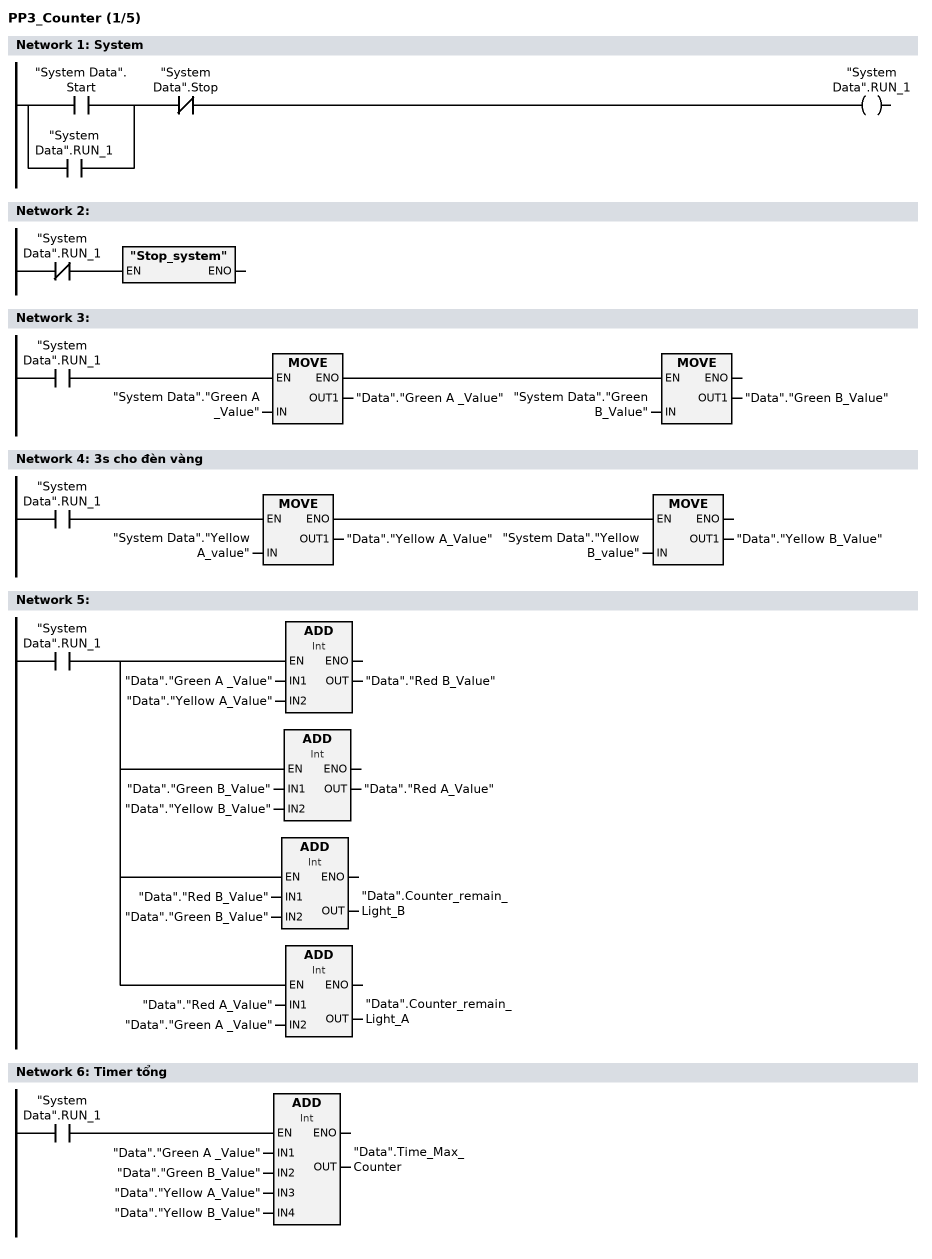
   RUNG wire#powerrail
      Contact( "System Data".Start )
      wire#w1
      I_Contact( "System Data".Stop )
      Coil( "System Data".RUN_1 )
   END_RUNG
   RUNG wire#powerrail
      Contact( "System Data".RUN_1 )
   END_RUNG wire#w1
   // the same network as SCL:
   "System Data".RUN_1 := ("System Data".Start OR "System Data".RUN_1) AND NOT "System Data".Stop;
END_REGION

REGION Network 2
   RUNG wire#powerrail
      I_Contact( "System Data".RUN_1 )
      "Stop_system"()
   END_RUNG
   // the same network as SCL:
   IF NOT "System Data".RUN_1 THEN "Stop_system"(); END_IF;
END_REGION

REGION Network 3
   RUNG wire#powerrail
      Contact( "System Data".RUN_1 )
      Move(in := "System Data"."Green A _Value", out1 => "Data"."Green A _Value")
      Move(in := "System Data"."Green B_Value", out1 => "Data"."Green B_Value")
   END_RUNG
   // the same network as SCL:
   IF "System Data".RUN_1 THEN
       "Data"."Green A _Value" := "System Data"."Green A _Value";
       "Data"."Green B_Value" := "System Data"."Green B_Value";
   END_IF;
END_REGION

REGION Network 4: 3s cho đèn vàng
   RUNG wire#powerrail
      Contact( "System Data".RUN_1 )
      Move(in := "System Data"."Yellow A_value", out1 => "Data"."Yellow A_Value")
      Move(in := "System Data"."Yellow B_value", out1 => "Data"."Yellow B_Value")
   END_RUNG
   // the same network as SCL:
   IF "System Data".RUN_1 THEN
       "Data"."Yellow A_Value" := "System Data"."Yellow A_value";
       "Data"."Yellow B_Value" := "System Data"."Yellow B_value";
   END_IF;
END_REGION

REGION Network 5
   RUNG wire#powerrail
      Contact( "System Data".RUN_1 )
      wire#w1
      { S7_Templates := "SrcType := Int" } Add(in1 := "Data"."Green A _Value", in2 := "Data"."Yellow A_Value", out => "Data"."Red B_Value")
   END_RUNG
   RUNG wire#w1
      { S7_Templates := "SrcType := Int" } Add(in1 := "Data"."Green B_Value", in2 := "Data"."Yellow B_Value", out => "Data"."Red A_Value")
   END_RUNG
   RUNG wire#w1
      { S7_Templates := "SrcType := Int" } Add(in1 := "Data"."Red B_Value", in2 := "Data"."Green B_Value", out => "Data".Counter_remain_Light_B)
   END_RUNG
   RUNG wire#w1
      { S7_Templates := "SrcType := Int" } Add(in1 := "Data"."Red A_Value", in2 := "Data"."Green A _Value", out => "Data".Counter_remain_Light_A)
   END_RUNG
   // the same network as SCL:
   IF "System Data".RUN_1 THEN
       "Data"."Red B_Value" := "Data"."Green A _Value" + "Data"."Yellow A_Value";
       "Data"."Red A_Value" := "Data"."Green B_Value" + "Data"."Yellow B_Value";
       "Data".Counter_remain_Light_B := "Data"."Red B_Value" + "Data"."Green B_Value";
       "Data".Counter_remain_Light_A := "Data"."Red A_Value" + "Data"."Green A _Value";
   END_IF;
END_REGION

REGION Network 6: Timer tổng
   RUNG wire#powerrail
      Contact( "System Data".RUN_1 )
      { S7_Templates := "SrcType := Int" } Add(in1 := "Data"."Green A _Value", in2 := "Data"."Green B_Value", in3 := "Data"."Yellow A_Value", in4 := "Data"."Yellow B_Value", out => "Data".Time_Max_Counter)
   END_RUNG
   // the same network as SCL:
   IF "System Data".RUN_1 THEN
       "Data".Time_Max_Counter := "Data"."Green A _Value" + "Data"."Green B_Value" + "Data"."Yellow A_Value" + "Data"."Yellow B_Value";
   END_IF;
END_REGION

REGION Network 7: Tạo xung 1s
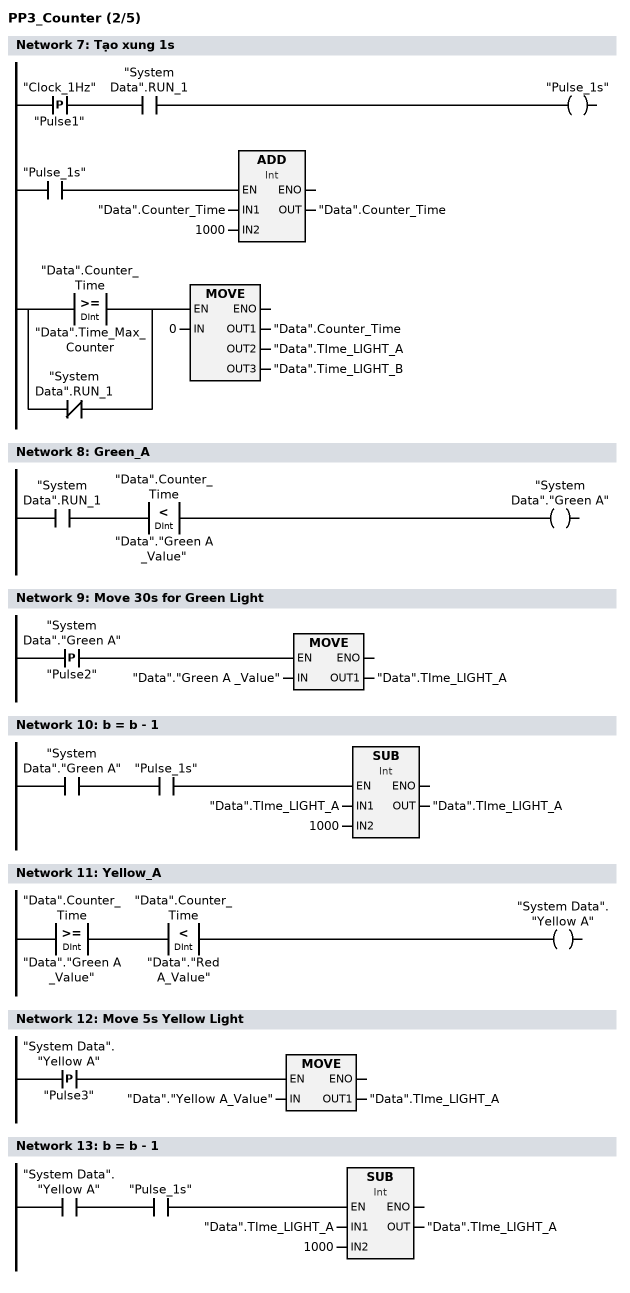
   RUNG wire#powerrail
      P_Contact(operand := "Clock_1Hz", bit := "Pulse1")
      Contact( "System Data".RUN_1 )
      Coil( "Pulse_1s" )
   END_RUNG
   RUNG wire#powerrail
      Contact( "Pulse_1s" )
      { S7_Templates := "SrcType := Int" } Add(in1 := "Data".Counter_Time, in2 := 1000, out => "Data".Counter_Time)
   END_RUNG
   RUNG wire#powerrail
      { S7_Templates := "SrcType := DInt" } GE_Contact(in1 := "Data".Counter_Time, in2 := "Data".Time_Max_Counter)
      wire#w1
      Move(in := 0, out1 => "Data".Counter_Time, out2 => "Data".TIme_LIGHT_A, out3 => "Data".Time_LIGHT_B)
   END_RUNG
   RUNG wire#powerrail
      I_Contact( "System Data".RUN_1 )
   END_RUNG wire#w1
   // the same network as SCL:
   #_w1 := "Clock_1Hz" AND NOT "Pulse1";   // rising edge of "Clock_1Hz"
   "Pulse1" := "Clock_1Hz";
   "Pulse_1s" := #_w1 AND "System Data".RUN_1;
   IF "Pulse_1s" THEN "Data".Counter_Time := "Data".Counter_Time + 1000; END_IF;
   IF ("Data".Counter_Time >= "Data".Time_Max_Counter) OR NOT "System Data".RUN_1 THEN
       "Data".Counter_Time := 0;
       "Data".TIme_LIGHT_A := 0;
       "Data".Time_LIGHT_B := 0;
   END_IF;
END_REGION

REGION Network 8: Green_A
   RUNG wire#powerrail
      Contact( "System Data".RUN_1 )
      { S7_Templates := "SrcType := DInt" } LT_Contact(in1 := "Data".Counter_Time, in2 := "Data"."Green A _Value")
      Coil( "System Data"."Green A" )
   END_RUNG
   // the same network as SCL:
   "System Data"."Green A" := "System Data".RUN_1 AND ("Data".Counter_Time < "Data"."Green A _Value");
END_REGION

REGION Network 9: Move 30s for Green Light
   RUNG wire#powerrail
      P_Contact(operand := "System Data"."Green A", bit := "Pulse2")
      Move(in := "Data"."Green A _Value", out1 => "Data".TIme_LIGHT_A)
   END_RUNG
   // the same network as SCL:
   #_w1 := "System Data"."Green A" AND NOT "Pulse2";   // rising edge of "System Data"."Green A"
   "Pulse2" := "System Data"."Green A";
   IF #_w1 THEN "Data".TIme_LIGHT_A := "Data"."Green A _Value"; END_IF;
END_REGION

REGION Network 10: b = b - 1
   RUNG wire#powerrail
      Contact( "System Data"."Green A" )
      Contact( "Pulse_1s" )
      { S7_Templates := "SrcType := Int" } Sub(in1 := "Data".TIme_LIGHT_A, in2 := 1000, out => "Data".TIme_LIGHT_A)
   END_RUNG
   // the same network as SCL:
   IF "System Data"."Green A" AND "Pulse_1s" THEN "Data".TIme_LIGHT_A := "Data".TIme_LIGHT_A - 1000; END_IF;
END_REGION

REGION Network 11: Yellow_A
   RUNG wire#powerrail
      { S7_Templates := "SrcType := DInt" } GE_Contact(in1 := "Data".Counter_Time, in2 := "Data"."Green A _Value")
      { S7_Templates := "SrcType := DInt" } LT_Contact(in1 := "Data".Counter_Time, in2 := "Data"."Red A_Value")
      Coil( "System Data"."Yellow A" )
   END_RUNG
   // the same network as SCL:
   "System Data"."Yellow A" := ("Data".Counter_Time >= "Data"."Green A _Value") AND ("Data".Counter_Time < "Data"."Red A_Value");
END_REGION

REGION Network 12: Move 5s Yellow Light
   RUNG wire#powerrail
      P_Contact(operand := "System Data"."Yellow A", bit := "Pulse3")
      Move(in := "Data"."Yellow A_Value", out1 => "Data".TIme_LIGHT_A)
   END_RUNG
   // the same network as SCL:
   #_w1 := "System Data"."Yellow A" AND NOT "Pulse3";   // rising edge of "System Data"."Yellow A"
   "Pulse3" := "System Data"."Yellow A";
   IF #_w1 THEN "Data".TIme_LIGHT_A := "Data"."Yellow A_Value"; END_IF;
END_REGION

REGION Network 13: b = b - 1
   RUNG wire#powerrail
      Contact( "System Data"."Yellow A" )
      Contact( "Pulse_1s" )
      { S7_Templates := "SrcType := Int" } Sub(in1 := "Data".TIme_LIGHT_A, in2 := 1000, out => "Data".TIme_LIGHT_A)
   END_RUNG
   // the same network as SCL:
   IF "System Data"."Yellow A" AND "Pulse_1s" THEN "Data".TIme_LIGHT_A := "Data".TIme_LIGHT_A - 1000; END_IF;
END_REGION

REGION Network 14: Red_A
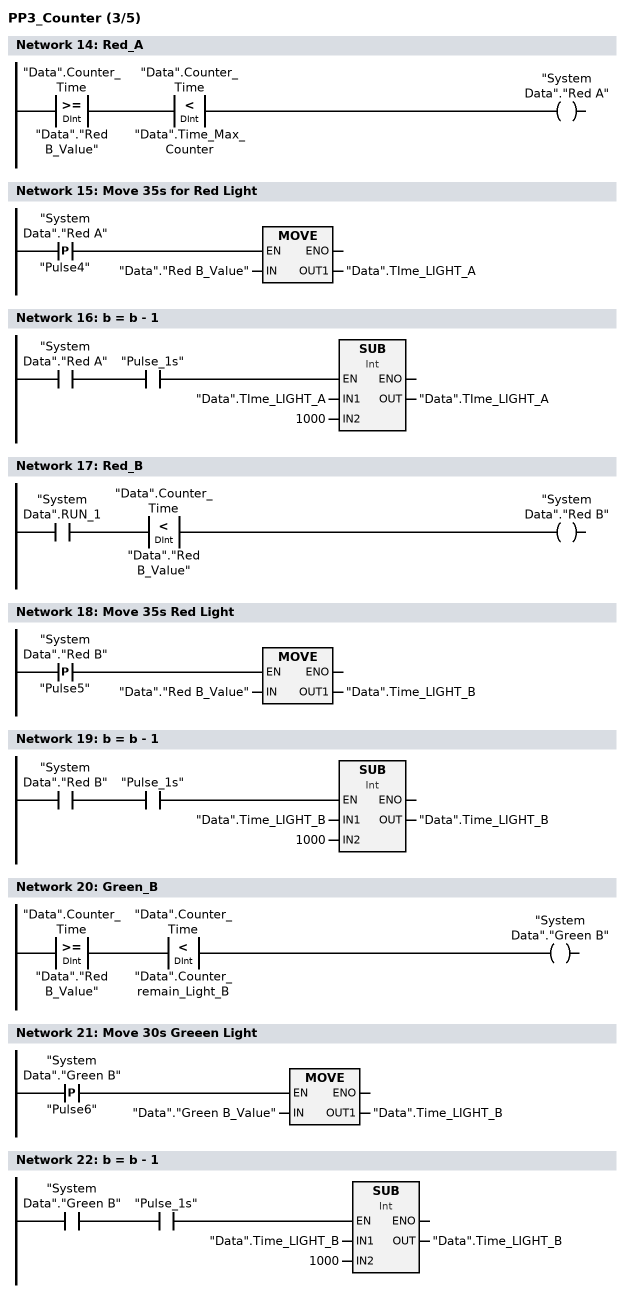
   RUNG wire#powerrail
      { S7_Templates := "SrcType := DInt" } GE_Contact(in1 := "Data".Counter_Time, in2 := "Data"."Red B_Value")
      { S7_Templates := "SrcType := DInt" } LT_Contact(in1 := "Data".Counter_Time, in2 := "Data".Time_Max_Counter)
      Coil( "System Data"."Red A" )
   END_RUNG
   // the same network as SCL:
   "System Data"."Red A" := ("Data".Counter_Time >= "Data"."Red B_Value") AND ("Data".Counter_Time < "Data".Time_Max_Counter);
END_REGION

REGION Network 15: Move 35s for Red Light
   RUNG wire#powerrail
      P_Contact(operand := "System Data"."Red A", bit := "Pulse4")
      Move(in := "Data"."Red B_Value", out1 => "Data".TIme_LIGHT_A)
   END_RUNG
   // the same network as SCL:
   #_w1 := "System Data"."Red A" AND NOT "Pulse4";   // rising edge of "System Data"."Red A"
   "Pulse4" := "System Data"."Red A";
   IF #_w1 THEN "Data".TIme_LIGHT_A := "Data"."Red B_Value"; END_IF;
END_REGION

REGION Network 16: b = b - 1
   RUNG wire#powerrail
      Contact( "System Data"."Red A" )
      Contact( "Pulse_1s" )
      { S7_Templates := "SrcType := Int" } Sub(in1 := "Data".TIme_LIGHT_A, in2 := 1000, out => "Data".TIme_LIGHT_A)
   END_RUNG
   // the same network as SCL:
   IF "System Data"."Red A" AND "Pulse_1s" THEN "Data".TIme_LIGHT_A := "Data".TIme_LIGHT_A - 1000; END_IF;
END_REGION

REGION Network 17: Red_B
   RUNG wire#powerrail
      Contact( "System Data".RUN_1 )
      { S7_Templates := "SrcType := DInt" } LT_Contact(in1 := "Data".Counter_Time, in2 := "Data"."Red B_Value")
      Coil( "System Data"."Red B" )
   END_RUNG
   // the same network as SCL:
   "System Data"."Red B" := "System Data".RUN_1 AND ("Data".Counter_Time < "Data"."Red B_Value");
END_REGION

REGION Network 18: Move 35s Red Light
   RUNG wire#powerrail
      P_Contact(operand := "System Data"."Red B", bit := "Pulse5")
      Move(in := "Data"."Red B_Value", out1 => "Data".Time_LIGHT_B)
   END_RUNG
   // the same network as SCL:
   #_w1 := "System Data"."Red B" AND NOT "Pulse5";   // rising edge of "System Data"."Red B"
   "Pulse5" := "System Data"."Red B";
   IF #_w1 THEN "Data".Time_LIGHT_B := "Data"."Red B_Value"; END_IF;
END_REGION

REGION Network 19: b = b - 1
   RUNG wire#powerrail
      Contact( "System Data"."Red B" )
      Contact( "Pulse_1s" )
      { S7_Templates := "SrcType := Int" } Sub(in1 := "Data".Time_LIGHT_B, in2 := 1000, out => "Data".Time_LIGHT_B)
   END_RUNG
   // the same network as SCL:
   IF "System Data"."Red B" AND "Pulse_1s" THEN "Data".Time_LIGHT_B := "Data".Time_LIGHT_B - 1000; END_IF;
END_REGION

REGION Network 20: Green_B
   RUNG wire#powerrail
      { S7_Templates := "SrcType := DInt" } GE_Contact(in1 := "Data".Counter_Time, in2 := "Data"."Red B_Value")
      { S7_Templates := "SrcType := DInt" } LT_Contact(in1 := "Data".Counter_Time, in2 := "Data".Counter_remain_Light_B)
      Coil( "System Data"."Green B" )
   END_RUNG
   // the same network as SCL:
   "System Data"."Green B" := ("Data".Counter_Time >= "Data"."Red B_Value") AND ("Data".Counter_Time < "Data".Counter_remain_Light_B);
END_REGION

REGION Network 21: Move 30s Greeen Light
   RUNG wire#powerrail
      P_Contact(operand := "System Data"."Green B", bit := "Pulse6")
      Move(in := "Data"."Green B_Value", out1 => "Data".Time_LIGHT_B)
   END_RUNG
   // the same network as SCL:
   #_w1 := "System Data"."Green B" AND NOT "Pulse6";   // rising edge of "System Data"."Green B"
   "Pulse6" := "System Data"."Green B";
   IF #_w1 THEN "Data".Time_LIGHT_B := "Data"."Green B_Value"; END_IF;
END_REGION

REGION Network 22: b = b - 1
   RUNG wire#powerrail
      Contact( "System Data"."Green B" )
      Contact( "Pulse_1s" )
      { S7_Templates := "SrcType := Int" } Sub(in1 := "Data".Time_LIGHT_B, in2 := 1000, out => "Data".Time_LIGHT_B)
   END_RUNG
   // the same network as SCL:
   IF "System Data"."Green B" AND "Pulse_1s" THEN "Data".Time_LIGHT_B := "Data".Time_LIGHT_B - 1000; END_IF;
END_REGION

REGION Network 23: Yellow_B
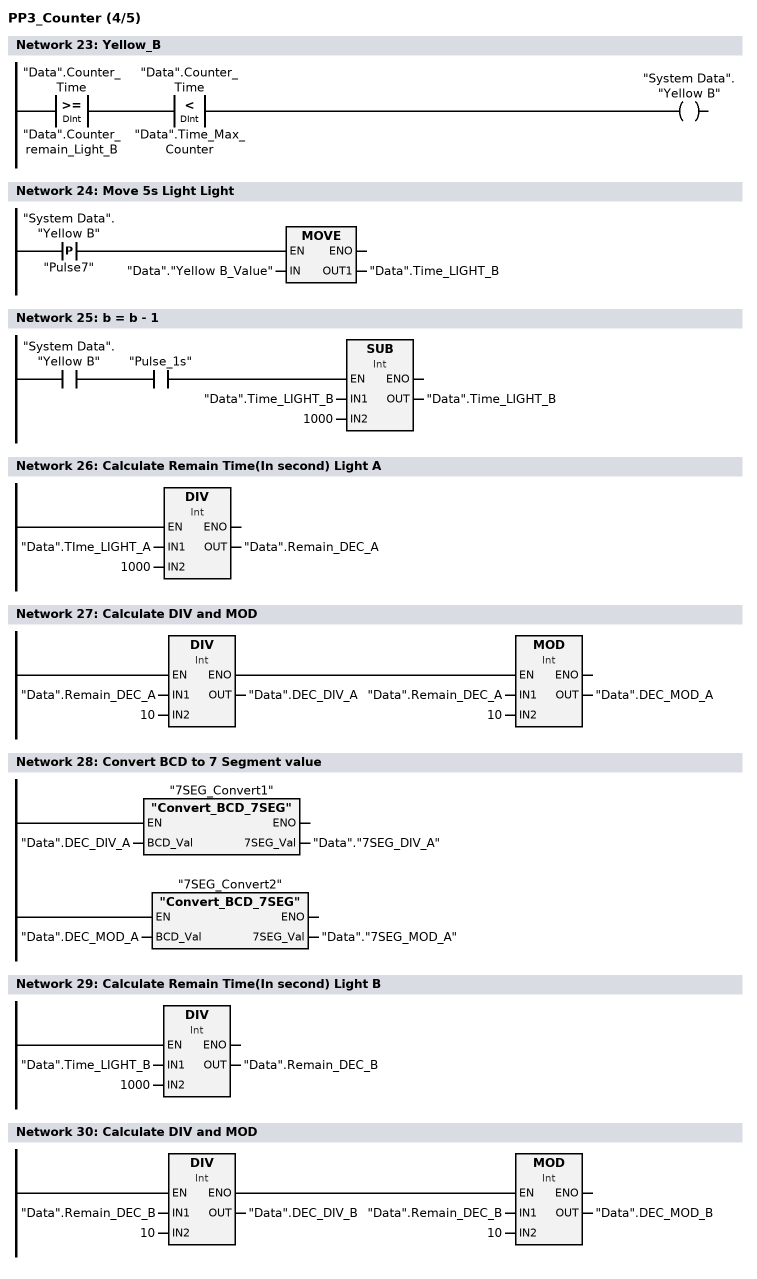
   RUNG wire#powerrail
      { S7_Templates := "SrcType := DInt" } GE_Contact(in1 := "Data".Counter_Time, in2 := "Data".Counter_remain_Light_B)
      { S7_Templates := "SrcType := DInt" } LT_Contact(in1 := "Data".Counter_Time, in2 := "Data".Time_Max_Counter)
      Coil( "System Data"."Yellow B" )
   END_RUNG
   // the same network as SCL:
   "System Data"."Yellow B" := ("Data".Counter_Time >= "Data".Counter_remain_Light_B) AND ("Data".Counter_Time < "Data".Time_Max_Counter);
END_REGION

REGION Network 24: Move 5s Light Light
   RUNG wire#powerrail
      P_Contact(operand := "System Data"."Yellow B", bit := "Pulse7")
      Move(in := "Data"."Yellow B_Value", out1 => "Data".Time_LIGHT_B)
   END_RUNG
   // the same network as SCL:
   #_w1 := "System Data"."Yellow B" AND NOT "Pulse7";   // rising edge of "System Data"."Yellow B"
   "Pulse7" := "System Data"."Yellow B";
   IF #_w1 THEN "Data".Time_LIGHT_B := "Data"."Yellow B_Value"; END_IF;
END_REGION

REGION Network 25: b = b - 1
   RUNG wire#powerrail
      Contact( "System Data"."Yellow B" )
      Contact( "Pulse_1s" )
      { S7_Templates := "SrcType := Int" } Sub(in1 := "Data".Time_LIGHT_B, in2 := 1000, out => "Data".Time_LIGHT_B)
   END_RUNG
   // the same network as SCL:
   IF "System Data"."Yellow B" AND "Pulse_1s" THEN "Data".Time_LIGHT_B := "Data".Time_LIGHT_B - 1000; END_IF;
END_REGION

REGION Network 26: Calculate Remain Time(In second) Light A
   RUNG wire#powerrail
      { S7_Templates := "SrcType := Int" } Div(in1 := "Data".TIme_LIGHT_A, in2 := 1000, out => "Data".Remain_DEC_A)
   END_RUNG
   // the same network as SCL:
   "Data".Remain_DEC_A := "Data".TIme_LIGHT_A / 1000;
END_REGION

REGION Network 27: Calculate DIV and MOD
   RUNG wire#powerrail
      { S7_Templates := "SrcType := Int" } Div(in1 := "Data".Remain_DEC_A, in2 := 10, out => "Data".DEC_DIV_A)
      { S7_Templates := "SrcType := Int" } Mod(in1 := "Data".Remain_DEC_A, in2 := 10, out => "Data".DEC_MOD_A)
   END_RUNG
   // the same network as SCL:
   "Data".DEC_DIV_A := "Data".Remain_DEC_A / 10;
   "Data".DEC_MOD_A := "Data".Remain_DEC_A MOD 10;
END_REGION

REGION Network 28: Convert BCD to 7 Segment value
   RUNG wire#powerrail
      "7SEG_Convert1"(BCD_Val := "Data".DEC_DIV_A, "7SEG_Val" => "Data"."7SEG_DIV_A")
   END_RUNG
   RUNG wire#powerrail
      "7SEG_Convert2"(BCD_Val := "Data".DEC_MOD_A, "7SEG_Val" => "Data"."7SEG_MOD_A")
   END_RUNG
   // the same network as SCL:
   "7SEG_Convert1"(BCD_Val := "Data".DEC_DIV_A, "7SEG_Val" => "Data"."7SEG_DIV_A");   // "Convert_BCD_7SEG"
   "7SEG_Convert2"(BCD_Val := "Data".DEC_MOD_A, "7SEG_Val" => "Data"."7SEG_MOD_A");   // "Convert_BCD_7SEG"
END_REGION

REGION Network 29: Calculate Remain Time(In second) Light B
   RUNG wire#powerrail
      { S7_Templates := "SrcType := Int" } Div(in1 := "Data".Time_LIGHT_B, in2 := 1000, out => "Data".Remain_DEC_B)
   END_RUNG
   // the same network as SCL:
   "Data".Remain_DEC_B := "Data".Time_LIGHT_B / 1000;
END_REGION

REGION Network 30: Calculate DIV and MOD
   RUNG wire#powerrail
      { S7_Templates := "SrcType := Int" } Div(in1 := "Data".Remain_DEC_B, in2 := 10, out => "Data".DEC_DIV_B)
      { S7_Templates := "SrcType := Int" } Mod(in1 := "Data".Remain_DEC_B, in2 := 10, out => "Data".DEC_MOD_B)
   END_RUNG
   // the same network as SCL:
   "Data".DEC_DIV_B := "Data".Remain_DEC_B / 10;
   "Data".DEC_MOD_B := "Data".Remain_DEC_B MOD 10;
END_REGION

REGION Network 31: Convert BCD to 7 Segment value
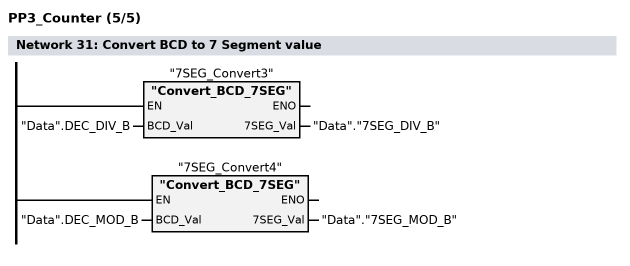
   RUNG wire#powerrail
      "7SEG_Convert3"(BCD_Val := "Data".DEC_DIV_B, "7SEG_Val" => "Data"."7SEG_DIV_B")
   END_RUNG
   RUNG wire#powerrail
      "7SEG_Convert4"(BCD_Val := "Data".DEC_MOD_B, "7SEG_Val" => "Data"."7SEG_MOD_B")
   END_RUNG
   // the same network as SCL:
   "7SEG_Convert3"(BCD_Val := "Data".DEC_DIV_B, "7SEG_Val" => "Data"."7SEG_DIV_B");   // "Convert_BCD_7SEG"
   "7SEG_Convert4"(BCD_Val := "Data".DEC_MOD_B, "7SEG_Val" => "Data"."7SEG_MOD_B");   // "Convert_BCD_7SEG"
END_REGION
END_FUNCTION

FUNCTION "Light_night" : Void   // FC4, LAD
{ S7_Optimized_Access := 'TRUE' }
VERSION : 0.1
BEGIN

REGION Network 1
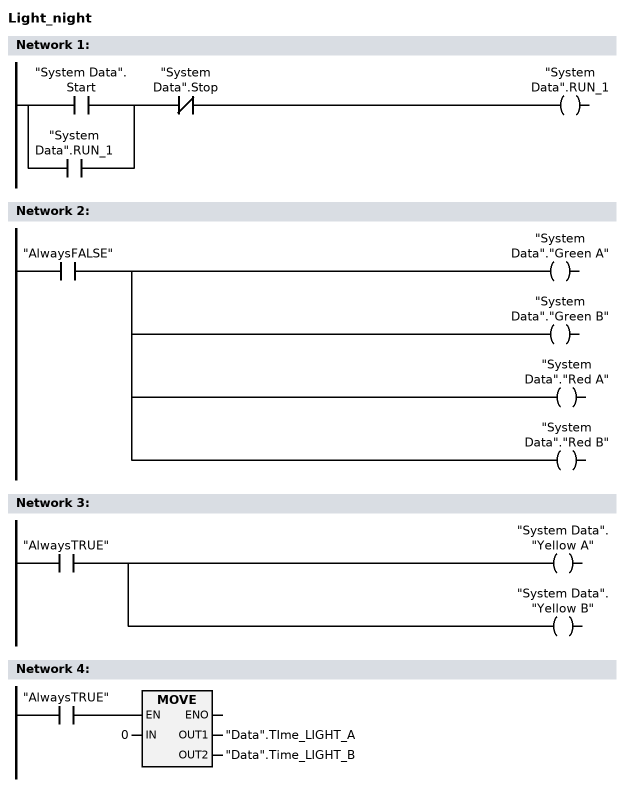
   RUNG wire#powerrail
      Contact( "System Data".Start )
      wire#w1
      I_Contact( "System Data".Stop )
      Coil( "System Data".RUN_1 )
   END_RUNG
   RUNG wire#powerrail
      Contact( "System Data".RUN_1 )
   END_RUNG wire#w1
   // the same network as SCL:
   "System Data".RUN_1 := ("System Data".Start OR "System Data".RUN_1) AND NOT "System Data".Stop;
END_REGION

REGION Network 2
   RUNG wire#powerrail
      Contact( "AlwaysFALSE" )
      wire#w1
      Coil( "System Data"."Green A" )
   END_RUNG
   RUNG wire#w1
      Coil( "System Data"."Green B" )
   END_RUNG
   RUNG wire#w1
      Coil( "System Data"."Red A" )
   END_RUNG
   RUNG wire#w1
      Coil( "System Data"."Red B" )
   END_RUNG
   // the same network as SCL:
   "System Data"."Green A" := "AlwaysFALSE";
   "System Data"."Green B" := "AlwaysFALSE";
   "System Data"."Red A" := "AlwaysFALSE";
   "System Data"."Red B" := "AlwaysFALSE";
END_REGION

REGION Network 3
   RUNG wire#powerrail
      Contact( "AlwaysTRUE" )
      wire#w1
      Coil( "System Data"."Yellow A" )
   END_RUNG
   RUNG wire#w1
      Coil( "System Data"."Yellow B" )
   END_RUNG
   // the same network as SCL:
   "System Data"."Yellow A" := "AlwaysTRUE";
   "System Data"."Yellow B" := "AlwaysTRUE";
END_REGION

REGION Network 4
   RUNG wire#powerrail
      Contact( "AlwaysTRUE" )
      Move(in := 0, out1 => "Data".TIme_LIGHT_A, out2 => "Data".Time_LIGHT_B)
   END_RUNG
   // the same network as SCL:
   IF "AlwaysTRUE" THEN
       "Data".TIme_LIGHT_A := 0;
       "Data".Time_LIGHT_B := 0;
   END_IF;
END_REGION
END_FUNCTION

FUNCTION "Function Local time" : Void   // FC5, LAD
{ S7_Optimized_Access := 'TRUE' }
VERSION : 0.1
BEGIN

REGION Network 1: Function read local time
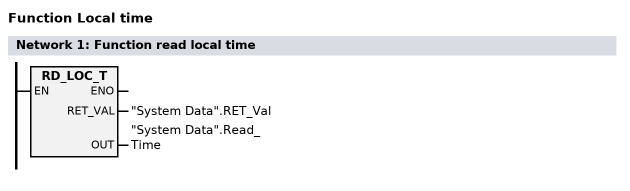
   "System Data".RET_Val := RD_LOC_T(OUT => "System Data".Read_Time);
END_REGION
END_FUNCTION

FUNCTION "Stop_system" : Void   // FC6, LAD
{ S7_Optimized_Access := 'TRUE' }
VERSION : 0.1
BEGIN

REGION Network 1
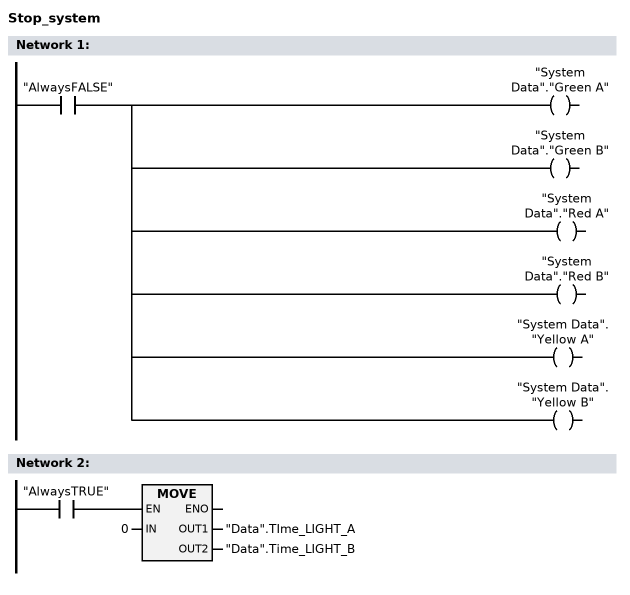
   RUNG wire#powerrail
      Contact( "AlwaysFALSE" )
      wire#w1
      Coil( "System Data"."Green A" )
   END_RUNG
   RUNG wire#w1
      Coil( "System Data"."Green B" )
   END_RUNG
   RUNG wire#w1
      Coil( "System Data"."Red A" )
   END_RUNG
   RUNG wire#w1
      Coil( "System Data"."Red B" )
   END_RUNG
   RUNG wire#w1
      Coil( "System Data"."Yellow A" )
   END_RUNG
   RUNG wire#w1
      Coil( "System Data"."Yellow B" )
   END_RUNG
   // the same network as SCL:
   "System Data"."Green A" := "AlwaysFALSE";
   "System Data"."Green B" := "AlwaysFALSE";
   "System Data"."Red A" := "AlwaysFALSE";
   "System Data"."Red B" := "AlwaysFALSE";
   "System Data"."Yellow A" := "AlwaysFALSE";
   "System Data"."Yellow B" := "AlwaysFALSE";
END_REGION

REGION Network 2
   RUNG wire#powerrail
      Contact( "AlwaysTRUE" )
      Move(in := 0, out1 => "Data".TIme_LIGHT_A, out2 => "Data".Time_LIGHT_B)
   END_RUNG
   // the same network as SCL:
   IF "AlwaysTRUE" THEN
       "Data".TIme_LIGHT_A := 0;
       "Data".Time_LIGHT_B := 0;
   END_IF;
END_REGION
END_FUNCTION

ORGANIZATION_BLOCK "Main"   // OB1, LAD, ProgramCycle
TITLE = "Main Program Sweep (Cycle)"
{ S7_Optimized_Access := 'TRUE' }
VERSION : 0.1
   VAR_INPUT
      Initial_Call : Bool;   // Initial call of this OB
      Remanence : Bool;   // =True, if remanent data are available
   END_VAR
   VAR_TEMP   // added for the SCL form of the ladder/FBD networks
      _w1 : Bool;
      _w2 : Bool;
      _w3 : Bool;
   END_VAR
BEGIN

REGION Network 1: Read local time
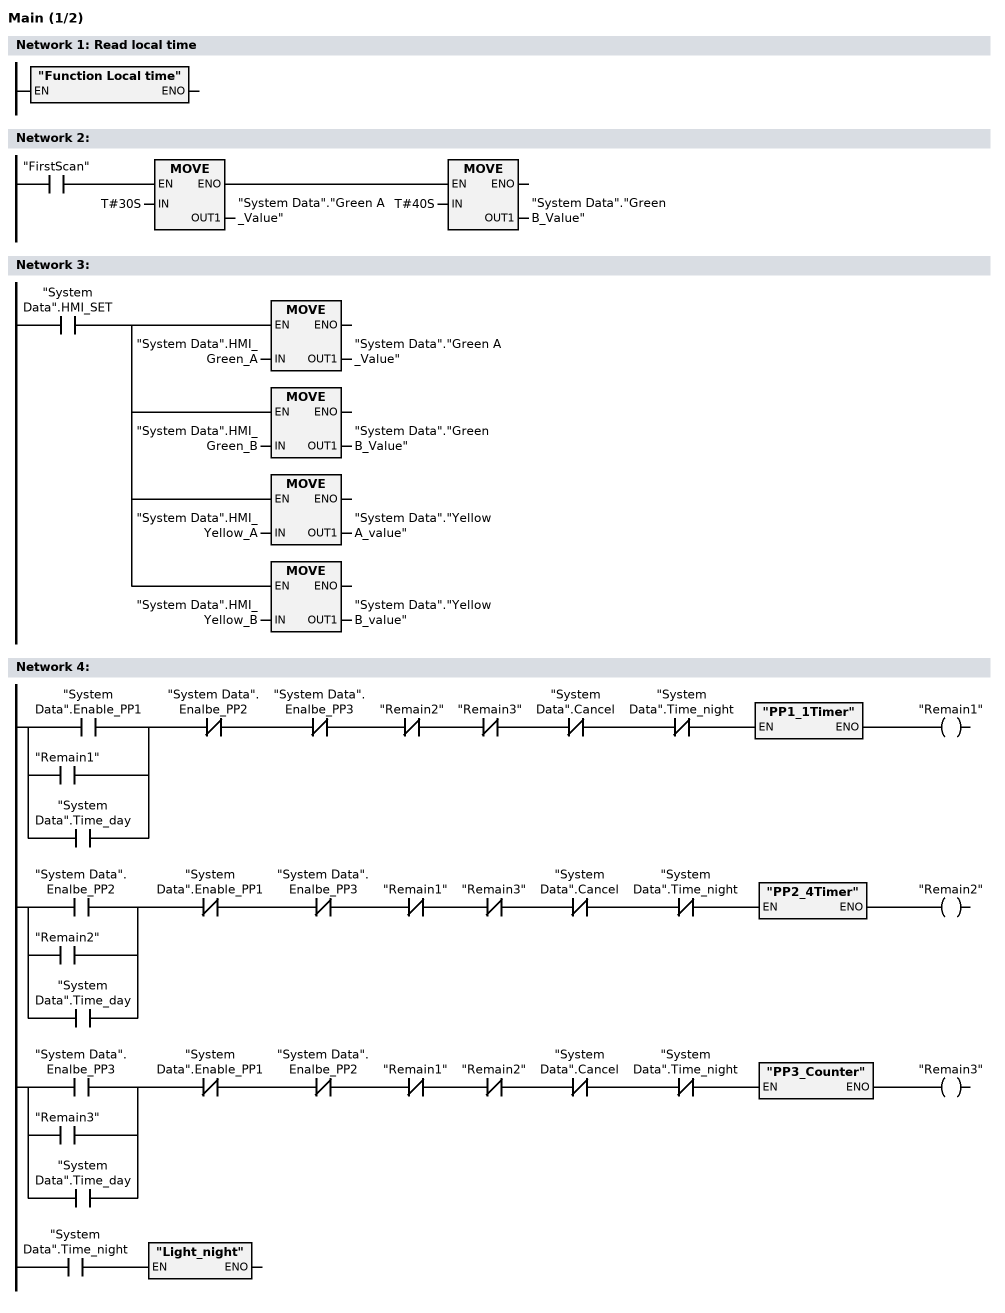
   RUNG wire#powerrail
      "Function Local time"()
   END_RUNG
   // the same network as SCL:
   "Function Local time"();
END_REGION

REGION Network 2
   RUNG wire#powerrail
      Contact( "FirstScan" )
      Move(in := T#30S, out1 => "System Data"."Green A _Value")
      Move(in := T#40S, out1 => "System Data"."Green B_Value")
   END_RUNG
   // the same network as SCL:
   IF "FirstScan" THEN
       "System Data"."Green A _Value" := T#30S;
       "System Data"."Green B_Value" := T#40S;
   END_IF;
END_REGION

REGION Network 3
   RUNG wire#powerrail
      Contact( "System Data".HMI_SET )
      wire#w1
      Move(in := "System Data".HMI_Green_A, out1 => "System Data"."Green A _Value")
   END_RUNG
   RUNG wire#w1
      Move(in := "System Data".HMI_Green_B, out1 => "System Data"."Green B_Value")
   END_RUNG
   RUNG wire#w1
      Move(in := "System Data".HMI_Yellow_A, out1 => "System Data"."Yellow A_value")
   END_RUNG
   RUNG wire#w1
      Move(in := "System Data".HMI_Yellow_B, out1 => "System Data"."Yellow B_value")
   END_RUNG
   // the same network as SCL:
   IF "System Data".HMI_SET THEN
       "System Data"."Green A _Value" := "System Data".HMI_Green_A;
       "System Data"."Green B_Value" := "System Data".HMI_Green_B;
       "System Data"."Yellow A_value" := "System Data".HMI_Yellow_A;
       "System Data"."Yellow B_value" := "System Data".HMI_Yellow_B;
   END_IF;
END_REGION

REGION Network 4
   RUNG wire#powerrail
      Contact( "System Data".Enable_PP1 )
      wire#w1
      I_Contact( "System Data".Enalbe_PP2 )
      I_Contact( "System Data".Enalbe_PP3 )
      I_Contact( "Remain2" )
      I_Contact( "Remain3" )
      I_Contact( "System Data".Cancel )
      I_Contact( "System Data".Time_night )
      "PP1_1Timer"()
      Coil( "Remain1" )
   END_RUNG
   RUNG wire#powerrail
      Contact( "Remain1" )
   END_RUNG wire#w1
   RUNG wire#powerrail
      Contact( "System Data".Time_day )
   END_RUNG wire#w1
   RUNG wire#powerrail
      Contact( "System Data".Enalbe_PP2 )
      wire#w2
      I_Contact( "System Data".Enable_PP1 )
      I_Contact( "System Data".Enalbe_PP3 )
      I_Contact( "Remain1" )
      I_Contact( "Remain3" )
      I_Contact( "System Data".Cancel )
      I_Contact( "System Data".Time_night )
      "PP2_4Timer"()
      Coil( "Remain2" )
   END_RUNG
   RUNG wire#powerrail
      Contact( "Remain2" )
   END_RUNG wire#w2
   RUNG wire#powerrail
      Contact( "System Data".Time_day )
   END_RUNG wire#w2
   RUNG wire#powerrail
      Contact( "System Data".Enalbe_PP3 )
      wire#w3
      I_Contact( "System Data".Enable_PP1 )
      I_Contact( "System Data".Enalbe_PP2 )
      I_Contact( "Remain1" )
      I_Contact( "Remain2" )
      I_Contact( "System Data".Cancel )
      I_Contact( "System Data".Time_night )
      "PP3_Counter"()
      Coil( "Remain3" )
   END_RUNG
   RUNG wire#powerrail
      Contact( "Remain3" )
   END_RUNG wire#w3
   RUNG wire#powerrail
      Contact( "System Data".Time_day )
   END_RUNG wire#w3
   RUNG wire#powerrail
      Contact( "System Data".Time_night )
      "Light_night"()
   END_RUNG
   // the same network as SCL:
   "PP1_1Timer"(EN := ("System Data".Enable_PP1 OR "Remain1" OR "System Data".Time_day) AND NOT "System Data".Enalbe_PP2 AND NOT "System Data".Enalbe_PP3 AND NOT "Remain2" AND NOT "Remain3" AND NOT "System Data".Cancel AND NOT "System Data".Time_night,
                ENO => #_w1);
   "Remain1" := #_w1;
   "PP2_4Timer"(EN := ("System Data".Enalbe_PP2 OR "Remain2" OR "System Data".Time_day) AND NOT "System Data".Enable_PP1 AND NOT "System Data".Enalbe_PP3 AND NOT "Remain1" AND NOT "Remain3" AND NOT "System Data".Cancel AND NOT "System Data".Time_night,
                ENO => #_w2);
   "Remain2" := #_w2;
   "PP3_Counter"(EN := ("System Data".Enalbe_PP3 OR "Remain3" OR "System Data".Time_day) AND NOT "System Data".Enable_PP1 AND NOT "System Data".Enalbe_PP2 AND NOT "Remain1" AND NOT "Remain2" AND NOT "System Data".Cancel AND NOT "System Data".Time_night,
                 ENO => #_w3);
   "Remain3" := #_w3;
   IF "System Data".Time_night THEN "Light_night"(); END_IF;
END_REGION

REGION Network 5: Day
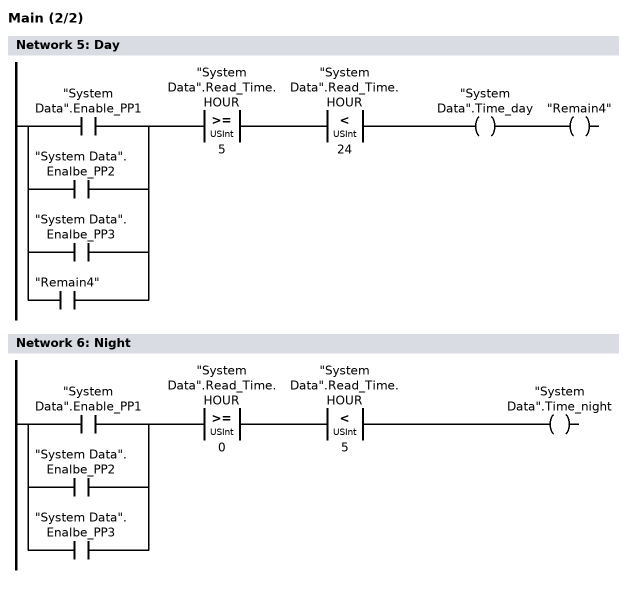
   RUNG wire#powerrail
      Contact( "System Data".Enable_PP1 )
      wire#w1
      { S7_Templates := "SrcType := USInt" } GE_Contact(in1 := "System Data".Read_Time.HOUR, in2 := 5)
      { S7_Templates := "SrcType := USInt" } LT_Contact(in1 := "System Data".Read_Time.HOUR, in2 := 24)
      Coil( "System Data".Time_day )
      Coil( "Remain4" )
   END_RUNG
   RUNG wire#powerrail
      Contact( "System Data".Enalbe_PP2 )
   END_RUNG wire#w1
   RUNG wire#powerrail
      Contact( "System Data".Enalbe_PP3 )
   END_RUNG wire#w1
   RUNG wire#powerrail
      Contact( "Remain4" )
   END_RUNG wire#w1
   // the same network as SCL:
   "System Data".Time_day := ("System Data".Enable_PP1 OR "System Data".Enalbe_PP2 OR "System Data".Enalbe_PP3 OR "Remain4") AND ("System Data".Read_Time.HOUR >= 5) AND ("System Data".Read_Time.HOUR < 24);
   "Remain4" := "System Data".Time_day;
END_REGION

REGION Network 6: Night
   RUNG wire#powerrail
      Contact( "System Data".Enable_PP1 )
      wire#w1
      { S7_Templates := "SrcType := USInt" } GE_Contact(in1 := "System Data".Read_Time.HOUR, in2 := 0)
      { S7_Templates := "SrcType := USInt" } LT_Contact(in1 := "System Data".Read_Time.HOUR, in2 := 5)
      Coil( "System Data".Time_night )
   END_RUNG
   RUNG wire#powerrail
      Contact( "System Data".Enalbe_PP2 )
   END_RUNG wire#w1
   RUNG wire#powerrail
      Contact( "System Data".Enalbe_PP3 )
   END_RUNG wire#w1
   // the same network as SCL:
   "System Data".Time_night := ("System Data".Enable_PP1 OR "System Data".Enalbe_PP2 OR "System Data".Enalbe_PP3) AND ("System Data".Read_Time.HOUR >= 0) AND ("System Data".Read_Time.HOUR < 5);
END_REGION
END_ORGANIZATION_BLOCK

(* ===== HMI "HMI_RT_1" =====
system functions are stored by id; their names below are inferred from use
connection "HMI_Connection_1": ETHERNET, SMART_S7_1200_OMS

HMI tags "Default tag table"
   "Tag_ScreenNumber" : UInt, internal

Template "Template_1" 800x480
   Button "Exit" at 714,429 size 71x50; TextOff 'Exit'; PictureOff "ExitRuntime_KTP700_Basic_PN_TR"; PictureOn "ExitRuntime_KTP700_Basic_PN_TR"
      on Release: StopRuntime(0)
   Button "Template_Button" at 614,429 size 71x50; TextOff 'Text'
   Button "Template_Button_1" at 514,429 size 71x50; TextOff 'Text'
   Button "Template_Button_2" at 414,429 size 71x50; TextOff 'Text'
   Button "Template_Button_3" at 314,429 size 71x50; TextOff 'Text'
   Button "Template_Button_4" at 214,429 size 71x50; TextOff 'Text'
   Button "Alarms" at 114,429 size 71x50; TextOff 'Alarms'; PictureOff "AlarmDisplay_KTP700_Basic_PN_TR"; PictureOn "AlarmDisplay_KTP700_Basic_PN_TR"
      on Release: function_ef3f5d25("Alarm window_Unacknowledged", -1)
   Button "Start screen" at 14,429 size 71x50; TextOff 'Start screen'; PictureOff "NavigateHome_KTP700_Basic_PN_TR"; PictureOn "NavigateHome_KTP700_Basic_PN_TR"
      on Release: ActivateScreen("Root screen", 0)
   SymbolicIOField "Symbolic_IO_Field_Screen" at 93,9 size 600x33; TextOff '0'; TextOn '1'; TextList "TextList_ScreenNames"
      ProcessValue <- "Tag_ScreenNumber"
      on Change: ActivateScreenByNumber("Tag_ScreenNumber", 0)
   DateTimeField "HmiScreenItemData" at 695,25 size 105x25
   DateTimeField "HmiScreenItemData_1" at 695,0 size 105x25
   GraphicView "Logo" at 0,0 size 91x51; Picture "Logo of HMI_1"

screen "Root screen" 800x480, template "Template_1"
   on GenerateScreen: SetTag("Tag_ScreenNumber", 1)
*)

(* ===== HMI "HMI_RT_2" =====
system functions are stored by id; their names below are inferred from use
connection "HMI_Connection_2": ETHERNET, S7_1200_OMS

HMI tags "Default tag table"
   "System Data_Green A" : Bool = PLC "System Data"."Green A", 1 s
   "System Data_Yellow A" : Bool = PLC "System Data"."Yellow A", 1 s
   "System Data_Red A" : Bool = PLC "System Data"."Red A", 1 s
   "System Data_Green B" : Bool = PLC "System Data"."Green B", 1 s
   "System Data_Yellow B" : Bool = PLC "System Data"."Yellow B", 1 s
   "System Data_Red B" : Bool = PLC "System Data"."Red B", 1 s
   "System Data_Start" : Bool = PLC "System Data".Start, 1 s
   "Timer1_ET" : Time = PLC Timer1.ET, 1 s
   "Timer2_ET" : Time = PLC Timer2.ET, 1 s
   "Timer3_ET" : Time = PLC Timer3.ET, 1 s
   "Timer4_Q" : Bool = PLC Timer4.Q, 1 s
   "Timer4_ET" : Time = PLC Timer4.ET, 1 s
   "System_Data_1timer_1Timer_TImer" : DInt = PLC Data.1Timer_TImer, 1 s
   "System Data_Green A _Value" : DInt = PLC "System Data"."Green A _Value", 1 s
   "System Data_Green B_Value" : DInt = PLC "System Data"."Green B_Value", 1 s
   "System Data_HMI_SET" : Bool = PLC "System Data".HMI_SET, 1 s
   "System Data_HMI_Green_A" : DInt = PLC "System Data".HMI_Green_A, 1 s
   "System Data_HMI_Green_B" : DInt = PLC "System Data".HMI_Green_B, 1 s
   "System Data_Stop" : Bool = PLC "System Data".Stop, 1 s
   "T1_ET" : Time = PLC T1.ET, 1 s
   "System_Data_1timer_TIme_Green_A" : DInt = PLC Data.TIme_LIGHT_A, 1 s
   "System_Data_1timer_Time_LIGHT_B" : DInt = PLC Data.Time_LIGHT_B, 1 s
   "System Data_Enable_PP1" : Bool = PLC "System Data".Enable_PP1, 1 s
   "System Data_Enalbe_PP2" : Bool = PLC "System Data".Enalbe_PP2, 1 s
   "System Data_Cancel" : Bool = PLC "System Data".Cancel, 1 s
   "System Data_Enalbe_PP3" : Bool = PLC "System Data".Enalbe_PP3, 1 s
   "System Data_HMI_Yellow_A" : DInt = PLC "System Data".HMI_Yellow_A, 1 s
   "System Data_HMI_Yellow_B" : DInt = PLC "System Data".HMI_Yellow_B, 1 s
   "Data_Timer_Red A_Value" : DInt = PLC Data."Red A_Value", 1 s
   "Data_Timer_Red B_Value" : DInt = PLC Data."Red B_Value", 1 s
   "Data_7SEG_DIV" : Byte = PLC Data.7SEG_DIV_A, 1 s
   "Data_7SEG_MOD" : Byte = PLC Data.7SEG_MOD_A, 1 s
   "Data_7SEG_DIV_B" : Byte = PLC Data.7SEG_DIV_B, 1 s
   "Data_7SEG_MOD_B" : Byte = PLC Data.7SEG_MOD_B, 1 s

screen "Screen_1" 1024x768
   Circle "Circle_1" at 176,128 size 48x48
      Appearance <- "System Data_Green A"
   Circle "Circle_2" at 176,201 size 48x48
      Appearance <- "System Data_Yellow A"
   Circle "Circle_3" at 176,274 size 48x48
      Appearance <- "System Data_Red A"
   Circle "Circle_4" at 296,128 size 48x48
      Appearance <- "System Data_Green B"
   Circle "Circle_5" at 296,201 size 48x48
      Appearance <- "System Data_Yellow B"
   Circle "Circle_6" at 296,274 size 48x48
      Appearance <- "System Data_Red B"
   IOField "I/O field_3" at 544,136 size 76x32; FormatPattern 99
      ProcessValue <- "System Data_HMI_Green_A"
   IOField "I/O field_4" at 544,176 size 76x32; FormatPattern 99
      ProcessValue <- "System Data_HMI_Yellow_A"
   IOField "I/O field_5" at 544,217 size 76x32; FormatPattern 99
      ProcessValue <- "Data_Timer_Red A_Value"
   Button "Button_3" at 740,294 size 68x32; TextOff 'SET'
      on Press: SetBit("System Data_HMI_SET")
      on Release: ResetBit("System Data_HMI_SET")
   Button "Button_1" at 465,293 size 61x32; TextOff 'Start'
      on Press: SetBit("System Data_Start")
      on Release: ResetBit("System Data_Start")
   Button "Button_4" at 526,293 size 56x32; TextOff 'Cancel'
      on Press: SetBit("System Data_Stop")
      on Release: ResetBit("System Data_Stop")
   IOField "I/O field_7" at 155,84 size 98x32; FormatPattern 99
      ProcessValue <- "System_Data_1timer_TIme_Green_A"
   IOField "I/O field_8" at 278,86 size 99x32; FormatPattern 99
      ProcessValue <- "System_Data_1timer_Time_LIGHT_B"
   Button "Button_2" at 498,331 size 96x32; TextOff '4Timer'
      on Press: SetBit("System Data_Enable_PP1")
      on Release: ResetBit("System Data_Enable_PP1")
      Appearance <- "System Data_Enable_PP1"
   Button "Button_5" at 606,331 size 96x32; TextOff '1 Timer'
      on Press: SetBit("System Data_Enalbe_PP2")
      on Release: ResetBit("System Data_Enalbe_PP2")
      Appearance <- "System Data_Enalbe_PP2"
   Button "Button_7" at 712,332 size 96x32; TextOff 'Counter'
      on Press: SetBit("System Data_Enalbe_PP3")
      on Release: ResetBit("System Data_Enalbe_PP3")
      Appearance <- "System Data_Enalbe_PP3"
   TextField "Text field_1" at 176,347 size 63x29; Text 'Side A'
   TextField "Text field_2" at 296,348 size 64x30; Text 'Side B'
   TextField "Text field_3" at 474,118 size 63x29; Text 'Side A'
   IOField "I/O field_9" at 710,136 size 76x32; FormatPattern 99
      ProcessValue <- "System Data_HMI_Green_B"
   IOField "I/O field_10" at 710,176 size 76x32; FormatPattern 99
      ProcessValue <- "System Data_HMI_Yellow_B"
   IOField "I/O field_11" at 710,217 size 76x32; FormatPattern 99
      ProcessValue <- "Data_Timer_Red B_Value"
   TextField "Text field_4" at 640,118 size 63x29; Text 'Side B'
   TextField "Text field_5" at 482,139 size 63x29; Text 'Green'
   TextField "Text field_6" at 482,176 size 63x29; Text 'Yellow'
   TextField "Text field_7" at 482,213 size 63x29; Text 'Red'
   TextField "Text field_8" at 647,136 size 63x29; Text 'Green'
   TextField "Text field_9" at 647,176 size 63x29; Text 'Yellow'
   TextField "Text field_10" at 647,216 size 63x29; Text 'Red'
   Rectangle "Rectangle_6" at 135,405 size 81x23
      Appearance <- "Data_7SEG_DIV"
   Rectangle "Rectangle_7" at 215,428 size 23x64
      Appearance <- "Data_7SEG_DIV"
   Rectangle "Rectangle_8" at 135,492 size 81x23
      Appearance <- "Data_7SEG_DIV"
   Rectangle "Rectangle_9" at 216,515 size 23x64
      Appearance <- "Data_7SEG_DIV"
   Rectangle "Rectangle_10" at 135,582 size 81x23
      Appearance <- "Data_7SEG_DIV"
   Rectangle "Rectangle_11" at 112,518 size 23x64
      Appearance <- "Data_7SEG_DIV"
   Rectangle "Rectangle_12" at 112,428 size 23x64
      Appearance <- "Data_7SEG_DIV"
   Rectangle "Rectangle_13" at 276,408 size 81x23
      Appearance <- "Data_7SEG_MOD"
   Rectangle "Rectangle_14" at 356,431 size 23x64
      Appearance <- "Data_7SEG_MOD"
   Rectangle "Rectangle_16" at 276,495 size 81x23
      Appearance <- "Data_7SEG_MOD"
   Rectangle "Rectangle_17" at 357,518 size 23x64
      Appearance <- "Data_7SEG_MOD"
   Rectangle "Rectangle_18" at 276,585 size 81x23
      Appearance <- "Data_7SEG_MOD"
   Rectangle "Rectangle_19" at 253,521 size 23x64
      Appearance <- "Data_7SEG_MOD"
   Rectangle "Rectangle_20" at 253,431 size 23x64
      Appearance <- "Data_7SEG_MOD"
   Rectangle "Rectangle_22" at 527,405 size 81x23
      Appearance <- "Data_7SEG_DIV_B"
   Rectangle "Rectangle_23" at 607,428 size 23x64
      Appearance <- "Data_7SEG_DIV_B"
   Rectangle "Rectangle_24" at 527,492 size 81x23
      Appearance <- "Data_7SEG_DIV_B"
   Rectangle "Rectangle_25" at 608,515 size 23x64
      Appearance <- "Data_7SEG_DIV_B"
   Rectangle "Rectangle_26" at 527,582 size 81x23
      Appearance <- "Data_7SEG_DIV_B"
   Rectangle "Rectangle_27" at 504,518 size 23x64
      Appearance <- "Data_7SEG_DIV_B"
   Rectangle "Rectangle_28" at 504,428 size 23x64
      Appearance <- "Data_7SEG_DIV_B"
   Rectangle "Rectangle_29" at 668,408 size 81x23
      Appearance <- "Data_7SEG_MOD_B"
   Rectangle "Rectangle_30" at 748,431 size 23x64
      Appearance <- "Data_7SEG_MOD_B"
   Rectangle "Rectangle_31" at 668,495 size 81x23
      Appearance <- "Data_7SEG_MOD_B"
   Rectangle "Rectangle_32" at 749,518 size 23x64
      Appearance <- "Data_7SEG_MOD_B"
   Rectangle "Rectangle_33" at 668,585 size 81x23
      Appearance <- "Data_7SEG_MOD_B"
   Rectangle "Rectangle_34" at 645,521 size 23x64
      Appearance <- "Data_7SEG_MOD_B"
   Rectangle "Rectangle_35" at 645,431 size 23x64
      Appearance <- "Data_7SEG_MOD_B"
   TextField "Text field_11" at 213,626 size 63x29; Text 'Side A'
   TextField "Text field_12" at 608,625 size 64x30; Text 'Side B'
   TextField "Text field_13" at 171,49 size 257x22; Text 'Võ Quang Thanh Nghĩa - 1851093'
*)